	X =  113.445  mm,	Y =   -643.534  mm,	Z =   -257.195  mm,
	W =  90.000 deg,	P =   0.000 deg,	R =   90.000 deg
};
P[2098]{
   GP1:
	UF : 0, UT : 6,		CONFIG : 'N U T, 0, 0, 0',
	X =  119.284  mm,	Y =   -640.249  mm,	Z =   -256.987  mm,
	W =  90.000 deg,	P =   0.000 deg,	R =   90.000 deg
};
P[2099]{
   GP1:
	UF : 0, UT : 6,		CONFIG : 'N U T, 0, 0, 0',
	X =  120.353  mm,	Y =   -639.513  mm,	Z =   -257.274  mm,
	W =  90.000 deg,	P =   0.000 deg,	R =   90.000 deg
};
P[2100]{
   GP1:
	UF : 0, UT : 6,		CONFIG : 'N U T, 0, 0, 0',
	X =  122.366  mm,	Y =   -638.374  mm,	Z =   -257.215  mm,
	W =  90.000 deg,	P =   0.000 deg,	R =   90.000 deg
};
P[2101]{
   GP1:
	UF : 0, UT : 6,		CONFIG : 'N U T, 0, 0, 0',
	X =  125.303  mm,	Y =   -636.720  mm,	Z =   -257.116  mm,
	W =  90.000 deg,	P =   0.000 deg,	R =   90.000 deg
};
P[2102]{
   GP1:
	UF : 0, UT : 6,		CONFIG : 'N U T, 0, 0, 0',
	X =  126.391  mm,	Y =   -636.119  mm,	Z =   -257.049  mm,
	W =  90.000 deg,	P =   0.000 deg,	R =   90.000 deg
};
P[2103]{
   GP1:
	UF : 0, UT : 6,		CONFIG : 'N U T, 0, 0, 0',
	X =  128.149  mm,	Y =   -635.072  mm,	Z =   -257.125  mm,
	W =  90.000 deg,	P =   0.000 deg,	R =   90.000 deg
};
P[2104]{
   GP1:
	UF : 0, UT : 6,		CONFIG : 'N U T, 0, 0, 0',
	X =  129.405  mm,	Y =   -634.261  mm,	Z =   -257.337  mm,
	W =  90.000 deg,	P =   0.000 deg,	R =   90.000 deg
};
P[2105]{
   GP1:
	UF : 0, UT : 6,		CONFIG : 'N U T, 0, 0, 0',
	X =  133.642  mm,	Y =   -631.812  mm,	Z =   -257.340  mm,
	W =  90.000 deg,	P =   0.000 deg,	R =   90.000 deg
};
P[2106]{
   GP1:
	UF : 0, UT : 6,		CONFIG : 'N U T, 0, 0, 0',
	X =  134.817  mm,	Y =   -631.137  mm,	Z =   -257.334  mm,
	W =  90.000 deg,	P =   0.000 deg,	R =   90.000 deg
};
P[2107]{
   GP1:
	UF : 0, UT : 6,		CONFIG : 'N U T, 0, 0, 0',
	X =  135.600  mm,	Y =   -630.719  mm,	Z =   -257.251  mm,
	W =  90.000 deg,	P =   0.000 deg,	R =   90.000 deg
};
P[2108]{
   GP1:
	UF : 0, UT : 6,		CONFIG : 'N U T, 0, 0, 0',
	X =  138.719  mm,	Y =   -628.949  mm,	Z =   -257.176  mm,
	W =  90.000 deg,	P =   0.000 deg,	R =   90.000 deg
};
P[2109]{
   GP1:
	UF : 0, UT : 6,		CONFIG : 'N U T, 0, 0, 0',
	X =  140.494  mm,	Y =   -627.843  mm,	Z =   -257.374  mm,
	W =  90.000 deg,	P =   0.000 deg,	R =   90.000 deg
};
P[2110]{
   GP1:
	UF : 0, UT : 6,		CONFIG : 'N U T, 0, 0, 0',
	X =  144.879  mm,	Y =   -625.464  mm,	Z =   -257.003  mm,
	W =  90.000 deg,	P =   0.000 deg,	R =   90.000 deg
};
P[2111]{
   GP1:
	UF : 0, UT : 6,		CONFIG : 'N U T, 0, 0, 0',
	X =  147.744  mm,	Y =   -623.730  mm,	Z =   -257.195  mm,
	W =  90.000 deg,	P =   0.000 deg,	R =   90.000 deg
};
P[2112]{
   GP1:
	UF : 0, UT : 6,		CONFIG : 'N U T, 0, 0, 0',
	X =  149.698  mm,	Y =   -622.634  mm,	Z =   -257.116  mm,
	W =  90.000 deg,	P =   0.000 deg,	R =   90.000 deg
};
P[2113]{
   GP1:
	UF : 0, UT : 6,		CONFIG : 'N U T, 0, 0, 0',
	X =  150.518  mm,	Y =   -622.121  mm,	Z =   -257.214  mm,
	W =  90.000 deg,	P =   0.000 deg,	R =   90.000 deg
};
P[2114]{
   GP1:
	UF : 0, UT : 6,		CONFIG : 'N U T, 0, 0, 0',
	X =  158.347  mm,	Y =   -617.647  mm,	Z =   -257.099  mm,
	W =  90.000 deg,	P =   0.000 deg,	R =   90.000 deg
};
P[2115]{
   GP1:
	UF : 0, UT : 6,		CONFIG : 'N U T, 0, 0, 0',
	X =  159.078  mm,	Y =   -617.197  mm,	Z =   -257.167  mm,
	W =  90.000 deg,	P =   0.000 deg,	R =   90.000 deg
};
P[2116]{
   GP1:
	UF : 0, UT : 6,		CONFIG : 'N U T, 0, 0, 0',
	X =  160.223  mm,	Y =   -616.456  mm,	Z =   -257.362  mm,
	W =  90.000 deg,	P =   0.000 deg,	R =   90.000 deg
};
P[2117]{
   GP1:
	UF : 0, UT : 6,		CONFIG : 'N U T, 0, 0, 0',
	X =  164.521  mm,	Y =   -614.083  mm,	Z =   -257.100  mm,
	W =  90.000 deg,	P =   0.000 deg,	R =   90.000 deg
};
P[2118]{
   GP1:
	UF : 0, UT : 6,		CONFIG : 'N U T, 0, 0, 0',
	X =  165.339  mm,	Y =   -613.695  mm,	Z =   -256.893  mm,
	W =  90.000 deg,	P =   0.000 deg,	R =   90.000 deg
};
P[2119]{
   GP1:
	UF : 0, UT : 6,		CONFIG : 'N U T, 0, 0, 0',
	X =  166.021  mm,	Y =   -613.178  mm,	Z =   -257.192  mm,
	W =  90.000 deg,	P =   0.000 deg,	R =   90.000 deg
};
P[2120]{
   GP1:
	UF : 0, UT : 6,		CONFIG : 'N U T, 0, 0, 0',
	X =  167.713  mm,	Y =   -612.213  mm,	Z =   -257.164  mm,
	W =  90.000 deg,	P =   0.000 deg,	R =   90.000 deg
};
P[2121]{
   GP1:
	UF : 0, UT : 6,		CONFIG : 'N U T, 0, 0, 0',
	X =  168.696  mm,	Y =   -611.619  mm,	Z =   -257.228  mm,
	W =  90.000 deg,	P =   0.000 deg,	R =   90.000 deg
};
P[2122]{
   GP1:
	UF : 0, UT : 6,		CONFIG : 'N U T, 0, 0, 0',
	X =  169.593  mm,	Y =   -611.059  mm,	Z =   -257.330  mm,
	W =  90.000 deg,	P =   0.000 deg,	R =   90.000 deg
};
P[2123]{
   GP1:
	UF : 0, UT : 6,		CONFIG : 'N U T, 0, 0, 0',
	X =  173.846  mm,	Y =   -608.622  mm,	Z =   -257.287  mm,
	W =  90.000 deg,	P =   0.000 deg,	R =   90.000 deg
};
P[2124]{
   GP1:
	UF : 0, UT : 6,		CONFIG : 'N U T, 0, 0, 0',
	X =  176.233  mm,	Y =   -607.353  mm,	Z =   -257.021  mm,
	W =  90.000 deg,	P =   0.000 deg,	R =   90.000 deg
};
P[2125]{
   GP1:
	UF : 0, UT : 6,		CONFIG : 'N U T, 0, 0, 0',
	X =  179.420  mm,	Y =   -605.394  mm,	Z =   -257.307  mm,
	W =  90.000 deg,	P =   0.000 deg,	R =   90.000 deg
};
P[2126]{
   GP1:
	UF : 0, UT : 6,		CONFIG : 'N U T, 0, 0, 0',
	X =  181.261  mm,	Y =   -604.330  mm,	Z =   -257.311  mm,
	W =  90.000 deg,	P =   0.000 deg,	R =   90.000 deg
};
P[2127]{
   GP1:
	UF : 0, UT : 6,		CONFIG : 'N U T, 0, 0, 0',
	X =  181.963  mm,	Y =   -604.005  mm,	Z =   -257.115  mm,
	W =  90.000 deg,	P =   0.000 deg,	R =   90.000 deg
};
P[2128]{
   GP1:
	UF : 0, UT : 6,		CONFIG : 'N U T, 0, 0, 0',
	X =  184.189  mm,	Y =   -602.626  mm,	Z =   -257.343  mm,
	W =  90.000 deg,	P =   0.000 deg,	R =   90.000 deg
};
P[2129]{
   GP1:
	UF : 0, UT : 6,		CONFIG : 'N U T, 0, 0, 0',
	X =  185.609  mm,	Y =   -601.897  mm,	Z =   -257.124  mm,
	W =  90.000 deg,	P =   0.000 deg,	R =   90.000 deg
};
P[2130]{
   GP1:
	UF : 0, UT : 6,		CONFIG : 'N U T, 0, 0, 0',
	X =  188.140  mm,	Y =   -600.372  mm,	Z =   -257.276  mm,
	W =  90.000 deg,	P =   0.000 deg,	R =   90.000 deg
};
P[2131]{
   GP1:
	UF : 0, UT : 6,		CONFIG : 'N U T, 0, 0, 0',
	X =  191.589  mm,	Y =   -598.356  mm,	Z =   -257.335  mm,
	W =  90.000 deg,	P =   0.000 deg,	R =   90.000 deg
};
P[2132]{
   GP1:
	UF : 0, UT : 6,		CONFIG : 'N U T, 0, 0, 0',
	X =  194.057  mm,	Y =   -596.933  mm,	Z =   -257.332  mm,
	W =  90.000 deg,	P =   0.000 deg,	R =   90.000 deg
};
P[2133]{
   GP1:
	UF : 0, UT : 6,		CONFIG : 'N U T, 0, 0, 0',
	X =  196.582  mm,	Y =   -595.509  mm,	Z =   -257.251  mm,
	W =  90.000 deg,	P =   0.000 deg,	R =   90.000 deg
};
P[2134]{
   GP1:
	UF : 0, UT : 6,		CONFIG : 'N U T, 0, 0, 0',
	X =  198.130  mm,	Y =   -594.683  mm,	Z =   -257.086  mm,
	W =  90.000 deg,	P =   0.000 deg,	R =   90.000 deg
};
P[2135]{
   GP1:
	UF : 0, UT : 6,		CONFIG : 'N U T, 0, 0, 0',
	X =  199.824  mm,	Y =   -593.721  mm,	Z =   -257.048  mm,
	W =  90.000 deg,	P =   0.000 deg,	R =   90.000 deg
};
P[2136]{
   GP1:
	UF : 0, UT : 6,		CONFIG : 'N U T, 0, 0, 0',
	X =  201.772  mm,	Y =   -592.515  mm,	Z =   -257.244  mm,
	W =  90.000 deg,	P =   0.000 deg,	R =   90.000 deg
};
P[2137]{
   GP1:
	UF : 0, UT : 6,		CONFIG : 'N U T, 0, 0, 0',
	X =  203.247  mm,	Y =   -591.664  mm,	Z =   -257.241  mm,
	W =  90.000 deg,	P =   0.000 deg,	R =   90.000 deg
};
P[2138]{
   GP1:
	UF : 0, UT : 6,		CONFIG : 'N U T, 0, 0, 0',
	X =  207.750  mm,	Y =   -589.114  mm,	Z =   -257.121  mm,
	W =  90.000 deg,	P =   0.000 deg,	R =   90.000 deg
};
P[2139]{
   GP1:
	UF : 0, UT : 6,		CONFIG : 'N U T, 0, 0, 0',
	X =  208.446  mm,	Y =   -588.732  mm,	Z =   -257.070  mm,
	W =  90.000 deg,	P =   0.000 deg,	R =   90.000 deg
};
P[2140]{
   GP1:
	UF : 0, UT : 6,		CONFIG : 'N U T, 0, 0, 0',
	X =  210.025  mm,	Y =   -587.832  mm,	Z =   -257.044  mm,
	W =  90.000 deg,	P =   0.000 deg,	R =   90.000 deg
};
P[2141]{
   GP1:
	UF : 0, UT : 6,		CONFIG : 'N U T, 0, 0, 0',
	X =  212.669  mm,	Y =   -586.209  mm,	Z =   -257.278  mm,
	W =  90.000 deg,	P =   0.000 deg,	R =   90.000 deg
};
P[2142]{
   GP1:
	UF : 0, UT : 6,		CONFIG : 'N U T, 0, 0, 0',
	X =  214.485  mm,	Y =   -585.126  mm,	Z =   -257.361  mm,
	W =  90.000 deg,	P =   0.000 deg,	R =   90.000 deg
};
P[2143]{
   GP1:
	UF : 0, UT : 6,		CONFIG : 'N U T, 0, 0, 0',
	X =  215.341  mm,	Y =   -584.730  mm,	Z =   -257.123  mm,
	W =  90.000 deg,	P =   0.000 deg,	R =   90.000 deg
};
P[2144]{
   GP1:
	UF : 0, UT : 6,		CONFIG : 'N U T, 0, 0, 0',
	X =  218.567  mm,	Y =   -582.892  mm,	Z =   -257.063  mm,
	W =  90.000 deg,	P =   0.000 deg,	R =   90.000 deg
};
P[2145]{
   GP1:
	UF : 0, UT : 6,		CONFIG : 'N U T, 0, 0, 0',
	X =  223.016  mm,	Y =   -580.308  mm,	Z =   -257.100  mm,
	W =  90.000 deg,	P =   0.000 deg,	R =   90.000 deg
};
P[2146]{
   GP1:
	UF : 0, UT : 6,		CONFIG : 'N U T, 0, 0, 0',
	X =  223.666  mm,	Y =   -580.001  mm,	Z =   -256.933  mm,
	W =  90.000 deg,	P =   0.000 deg,	R =   90.000 deg
};
P[2147]{
   GP1:
	UF : 0, UT : 6,		CONFIG : 'N U T, 0, 0, 0',
	X =  226.605  mm,	Y =   -578.307  mm,	Z =   -256.925  mm,
	W =  90.000 deg,	P =   0.000 deg,	R =   90.000 deg
};
P[2148]{
   GP1:
	UF : 0, UT : 6,		CONFIG : 'N U T, 0, 0, 0',
	X =  228.043  mm,	Y =   -577.321  mm,	Z =   -257.304  mm,
	W =  90.000 deg,	P =   0.000 deg,	R =   90.000 deg
};
P[2149]{
   GP1:
	UF : 0, UT : 6,		CONFIG : 'N U T, 0, 0, 0',
	X =  228.786  mm,	Y =   -577.012  mm,	Z =   -257.013  mm,
	W =  90.000 deg,	P =   0.000 deg,	R =   90.000 deg
};
P[2150]{
   GP1:
	UF : 0, UT : 6,		CONFIG : 'N U T, 0, 0, 0',
	X =  232.019  mm,	Y =   -575.058  mm,	Z =   -257.225  mm,
	W =  90.000 deg,	P =   0.000 deg,	R =   90.000 deg
};
P[2151]{
   GP1:
	UF : 0, UT : 6,		CONFIG : 'N U T, 0, 0, 0',
	X =  232.928  mm,	Y =   -574.469  mm,	Z =   -257.381  mm,
	W =  90.000 deg,	P =   0.000 deg,	R =   90.000 deg
};
P[2152]{
   GP1:
	UF : 0, UT : 6,		CONFIG : 'N U T, 0, 0, 0',
	X =  235.660  mm,	Y =   -572.931  mm,	Z =   -257.286  mm,
	W =  90.000 deg,	P =   0.000 deg,	R =   90.000 deg
};
P[2153]{
   GP1:
	UF : 0, UT : 6,		CONFIG : 'N U T, 0, 0, 0',
	X =  237.324  mm,	Y =   -572.109  mm,	Z =   -256.947  mm,
	W =  90.000 deg,	P =   0.000 deg,	R =   90.000 deg
};
P[2154]{
   GP1:
	UF : 0, UT : 6,		CONFIG : 'N U T, 0, 0, 0',
	X =  238.722  mm,	Y =   -571.134  mm,	Z =   -257.357  mm,
	W =  90.000 deg,	P =   0.000 deg,	R =   90.000 deg
};
P[2155]{
   GP1:
	UF : 0, UT : 6,		CONFIG : 'N U T, 0, 0, 0',
	X =  242.232  mm,	Y =   -569.250  mm,	Z =   -257.009  mm,
	W =  90.000 deg,	P =   0.000 deg,	R =   90.000 deg
};
P[2156]{
   GP1:
	UF : 0, UT : 6,		CONFIG : 'N U T, 0, 0, 0',
	X =  244.183  mm,	Y =   -567.996  mm,	Z =   -257.322  mm,
	W =  90.000 deg,	P =   0.000 deg,	R =   90.000 deg
};
P[2157]{
   GP1:
	UF : 0, UT : 6,		CONFIG : 'N U T, 0, 0, 0',
	X =  245.455  mm,	Y =   -567.331  mm,	Z =   -257.152  mm,
	W =  90.000 deg,	P =   0.000 deg,	R =   90.000 deg
};
P[2158]{
   GP1:
	UF : 0, UT : 6,		CONFIG : 'N U T, 0, 0, 0',
	X =  246.314  mm,	Y =   -566.740  mm,	Z =   -257.380  mm,
	W =  90.000 deg,	P =   0.000 deg,	R =   90.000 deg
};
P[2159]{
   GP1:
	UF : 0, UT : 6,		CONFIG : 'N U T, 0, 0, 0',
	X =  247.191  mm,	Y =   -566.275  mm,	Z =   -257.279  mm,
	W =  90.000 deg,	P =   0.000 deg,	R =   90.000 deg
};
P[2160]{
   GP1:
	UF : 0, UT : 6,		CONFIG : 'N U T, 0, 0, 0',
	X =  248.158  mm,	Y =   -565.716  mm,	Z =   -257.281  mm,
	W =  90.000 deg,	P =   0.000 deg,	R =   90.000 deg
};
P[2161]{
   GP1:
	UF : 0, UT : 6,		CONFIG : 'N U T, 0, 0, 0',
	X =  250.314  mm,	Y =   -564.475  mm,	Z =   -257.271  mm,
	W =  90.000 deg,	P =   0.000 deg,	R =   90.000 deg
};
P[2162]{
   GP1:
	UF : 0, UT : 6,		CONFIG : 'N U T, 0, 0, 0',
	X =  251.403  mm,	Y =   -563.903  mm,	Z =   -257.135  mm,
	W =  90.000 deg,	P =   0.000 deg,	R =   90.000 deg
};
P[2163]{
   GP1:
	UF : 0, UT : 6,		CONFIG : 'N U T, 0, 0, 0',
	X =  253.414  mm,	Y =   -562.723  mm,	Z =   -257.183  mm,
	W =  90.000 deg,	P =   0.000 deg,	R =   90.000 deg
};
P[2164]{
   GP1:
	UF : 0, UT : 6,		CONFIG : 'N U T, 0, 0, 0',
	X =  259.113  mm,	Y =   -559.505  mm,	Z =   -257.004  mm,
	W =  90.000 deg,	P =   0.000 deg,	R =   90.000 deg
};
P[2165]{
   GP1:
	UF : 0, UT : 6,		CONFIG : 'N U T, 0, 0, 0',
	X =  261.683  mm,	Y =   -557.964  mm,	Z =   -257.143  mm,
	W =  90.000 deg,	P =   0.000 deg,	R =   90.000 deg
};
P[2166]{
   GP1:
	UF : 0, UT : 6,		CONFIG : 'N U T, 0, 0, 0',
	X =  262.661  mm,	Y =   -557.339  mm,	Z =   -257.291  mm,
	W =  90.000 deg,	P =   0.000 deg,	R =   90.000 deg
};
P[2167]{
   GP1:
	UF : 0, UT : 6,		CONFIG : 'N U T, 0, 0, 0',
	X =  263.771  mm,	Y =   -556.827  mm,	Z =   -256.978  mm,
	W =  90.000 deg,	P =   0.000 deg,	R =   90.000 deg
};
P[2168]{
   GP1:
	UF : 0, UT : 6,		CONFIG : 'N U T, 0, 0, 0',
	X =  266.090  mm,	Y =   -555.345  mm,	Z =   -257.325  mm,
	W =  90.000 deg,	P =   0.000 deg,	R =   90.000 deg
};
P[2169]{
   GP1:
	UF : 0, UT : 6,		CONFIG : 'N U T, 0, 0, 0',
	X =  266.938  mm,	Y =   -555.016  mm,	Z =   -256.934  mm,
	W =  90.000 deg,	P =   0.000 deg,	R =   90.000 deg
};
P[2170]{
   GP1:
	UF : 0, UT : 6,		CONFIG : 'N U T, 0, 0, 0',
	X =  270.560  mm,	Y =   -552.768  mm,	Z =   -257.316  mm,
	W =  90.000 deg,	P =   0.000 deg,	R =   90.000 deg
};
P[2171]{
   GP1:
	UF : 0, UT : 6,		CONFIG : 'N U T, 0, 0, 0',
	X =  272.010  mm,	Y =   -551.959  mm,	Z =   -257.248  mm,
	W =  90.000 deg,	P =   0.000 deg,	R =   90.000 deg
};
P[2172]{
   GP1:
	UF : 0, UT : 6,		CONFIG : 'N U T, 0, 0, 0',
	X =  273.469  mm,	Y =   -551.079  mm,	Z =   -257.337  mm,
	W =  90.000 deg,	P =   0.000 deg,	R =   90.000 deg
};
P[2173]{
   GP1:
	UF : 0, UT : 6,		CONFIG : 'N U T, 0, 0, 0',
	X =  277.285  mm,	Y =   -548.933  mm,	Z =   -257.198  mm,
	W =  90.000 deg,	P =   0.000 deg,	R =   90.000 deg
};
P[2174]{
   GP1:
	UF : 0, UT : 6,		CONFIG : 'N U T, 0, 0, 0',
	X =  280.570  mm,	Y =   -546.991  mm,	Z =   -257.309  mm,
	W =  90.000 deg,	P =   0.000 deg,	R =   90.000 deg
};
P[2175]{
   GP1:
	UF : 0, UT : 6,		CONFIG : 'N U T, 0, 0, 0',
	X =  282.214  mm,	Y =   -546.154  mm,	Z =   -257.036  mm,
	W =  90.000 deg,	P =   0.000 deg,	R =   90.000 deg
};
P[2176]{
   GP1:
	UF : 0, UT : 6,		CONFIG : 'N U T, 0, 0, 0',
	X =  284.085  mm,	Y =   -544.962  mm,	Z =   -257.306  mm,
	W =  90.000 deg,	P =   0.000 deg,	R =   90.000 deg
};
P[2177]{
   GP1:
	UF : 0, UT : 6,		CONFIG : 'N U T, 0, 0, 0',
	X =  286.474  mm,	Y =   -543.555  mm,	Z =   -257.373  mm,
	W =  90.000 deg,	P =   0.000 deg,	R =   90.000 deg
};
P[2178]{
   GP1:
	UF : 0, UT : 6,		CONFIG : 'N U T, 0, 0, 0',
	X =  288.966  mm,	Y =   -542.236  mm,	Z =   -257.081  mm,
	W =  90.000 deg,	P =   0.000 deg,	R =   90.000 deg
};
P[2179]{
   GP1:
	UF : 0, UT : 6,		CONFIG : 'N U T, 0, 0, 0',
	X =  292.153  mm,	Y =   -540.456  mm,	Z =   -256.936  mm,
	W =  90.000 deg,	P =   0.000 deg,	R =   90.000 deg
};
P[2180]{
   GP1:
	UF : 0, UT : 6,		CONFIG : 'N U T, 0, 0, 0',
	X =  299.062  mm,	Y =   -536.298  mm,	Z =   -257.346  mm,
	W =  90.000 deg,	P =   0.000 deg,	R =   90.000 deg
};
P[2181]{
   GP1:
	UF : 0, UT : 6,		CONFIG : 'N U T, 0, 0, 0',
	X =  299.968  mm,	Y =   -535.760  mm,	Z =   -257.381  mm,
	W =  90.000 deg,	P =   0.000 deg,	R =   90.000 deg
};
P[2182]{
   GP1:
	UF : 0, UT : 6,		CONFIG : 'N U T, 0, 0, 0',
	X =  300.824  mm,	Y =   -535.320  mm,	Z =   -257.251  mm,
	W =  90.000 deg,	P =   0.000 deg,	R =   90.000 deg
};
P[2183]{
   GP1:
	UF : 0, UT : 6,		CONFIG : 'N U T, 0, 0, 0',
	X =  301.911  mm,	Y =   -534.684  mm,	Z =   -257.272  mm,
	W =  90.000 deg,	P =   0.000 deg,	R =   90.000 deg
};
P[2184]{
   GP1:
	UF : 0, UT : 6,		CONFIG : 'N U T, 0, 0, 0',
	X =  305.019  mm,	Y =   -532.905  mm,	Z =   -257.233  mm,
	W =  90.000 deg,	P =   0.000 deg,	R =   90.000 deg
};
P[2185]{
   GP1:
	UF : 0, UT : 6,		CONFIG : 'N U T, 0, 0, 0',
	X =  307.325  mm,	Y =   -531.551  mm,	Z =   -257.287  mm,
	W =  90.000 deg,	P =   0.000 deg,	R =   90.000 deg
};
P[2186]{
   GP1:
	UF : 0, UT : 6,		CONFIG : 'N U T, 0, 0, 0',
	X =  309.546  mm,	Y =   -530.345  mm,	Z =   -257.103  mm,
	W =  90.000 deg,	P =   0.000 deg,	R =   90.000 deg
};
P[2187]{
   GP1:
	UF : 0, UT : 6,		CONFIG : 'N U T, 0, 0, 0',
	X =  311.447  mm,	Y =   -529.152  mm,	Z =   -257.334  mm,
	W =  90.000 deg,	P =   0.000 deg,	R =   90.000 deg
};
P[2188]{
   GP1:
	UF : 0, UT : 6,		CONFIG : 'N U T, 0, 0, 0',
	X =  314.729  mm,	Y =   -527.268  mm,	Z =   -257.306  mm,
	W =  90.000 deg,	P =   0.000 deg,	R =   90.000 deg
};
P[2189]{
   GP1:
	UF : 0, UT : 6,		CONFIG : 'N U T, 0, 0, 0',
	X =  316.875  mm,	Y =   -526.069  mm,	Z =   -257.211  mm,
	W =  90.000 deg,	P =   0.000 deg,	R =   90.000 deg
};
P[2190]{
   GP1:
	UF : 0, UT : 6,		CONFIG : 'N U T, 0, 0, 0',
	X =  318.015  mm,	Y =   -525.355  mm,	Z =   -257.345  mm,
	W =  90.000 deg,	P =   0.000 deg,	R =   90.000 deg
};
P[2191]{
   GP1:
	UF : 0, UT : 6,		CONFIG : 'N U T, 0, 0, 0',
	X =  318.649  mm,	Y =   -525.057  mm,	Z =   -257.180  mm,
	W =  90.000 deg,	P =   0.000 deg,	R =   90.000 deg
};
P[2192]{
   GP1:
	UF : 0, UT : 6,		CONFIG : 'N U T, 0, 0, 0',
	X =  322.343  mm,	Y =   -522.958  mm,	Z =   -257.099  mm,
	W =  90.000 deg,	P =   0.000 deg,	R =   90.000 deg
};
P[2193]{
   GP1:
	UF : 0, UT : 6,		CONFIG : 'N U T, 0, 0, 0',
	X =  322.941  mm,	Y =   -522.528  mm,	Z =   -257.305  mm,
	W =  90.000 deg,	P =   0.000 deg,	R =   90.000 deg
};
P[2194]{
   GP1:
	UF : 0, UT : 6,		CONFIG : 'N U T, 0, 0, 0',
	X =  324.717  mm,	Y =   -521.576  mm,	Z =   -257.127  mm,
	W =  90.000 deg,	P =   0.000 deg,	R =   90.000 deg
};
P[2195]{
   GP1:
	UF : 0, UT : 6,		CONFIG : 'N U T, 0, 0, 0',
	X =  327.318  mm,	Y =   -520.012  mm,	Z =   -257.277  mm,
	W =  90.000 deg,	P =   0.000 deg,	R =   90.000 deg
};
P[2196]{
   GP1:
	UF : 0, UT : 6,		CONFIG : 'N U T, 0, 0, 0',
	X =  329.668  mm,	Y =   -518.723  mm,	Z =   -257.112  mm,
	W =  90.000 deg,	P =   0.000 deg,	R =   90.000 deg
};
P[2197]{
   GP1:
	UF : 0, UT : 6,		CONFIG : 'N U T, 0, 0, 0',
	X =  331.747  mm,	Y =   -517.451  mm,	Z =   -257.286  mm,
	W =  90.000 deg,	P =   0.000 deg,	R =   90.000 deg
};
P[2198]{
   GP1:
	UF : 0, UT : 6,		CONFIG : 'N U T, 0, 0, 0',
	X =  335.566  mm,	Y =   -515.313  mm,	Z =   -257.124  mm,
	W =  90.000 deg,	P =   0.000 deg,	R =   90.000 deg
};
P[2199]{
   GP1:
	UF : 0, UT : 6,		CONFIG : 'N U T, 0, 0, 0',
	X =  337.324  mm,	Y =   -514.263  mm,	Z =   -257.209  mm,
	W =  90.000 deg,	P =   0.000 deg,	R =   90.000 deg
};
P[2200]{
   GP1:
	UF : 0, UT : 6,		CONFIG : 'N U T, 0, 0, 0',
	X =  338.434  mm,	Y =   -513.597  mm,	Z =   -257.269  mm,
	W =  90.000 deg,	P =   0.000 deg,	R =   90.000 deg
};
P[2201]{
   GP1:
	UF : 0, UT : 6,		CONFIG : 'N U T, 0, 0, 0',
	X =  340.084  mm,	Y =   -512.599  mm,	Z =   -257.377  mm,
	W =  90.000 deg,	P =   0.000 deg,	R =   90.000 deg
};
P[2202]{
   GP1:
	UF : 0, UT : 6,		CONFIG : 'N U T, 0, 0, 0',
	X =  342.231  mm,	Y =   -511.494  mm,	Z =   -257.053  mm,
	W =  90.000 deg,	P =   0.000 deg,	R =   90.000 deg
};
P[2203]{
   GP1:
	UF : 0, UT : 6,		CONFIG : 'N U T, 0, 0, 0',
	X =  344.018  mm,	Y =   -510.380  mm,	Z =   -257.251  mm,
	W =  90.000 deg,	P =   0.000 deg,	R =   90.000 deg
};
P[2204]{
   GP1:
	UF : 0, UT : 6,		CONFIG : 'N U T, 0, 0, 0',
	X =  346.852  mm,	Y =   -508.709  mm,	Z =   -257.335  mm,
	W =  90.000 deg,	P =   0.000 deg,	R =   90.000 deg
};
P[2205]{
   GP1:
	UF : 0, UT : 6,		CONFIG : 'N U T, 0, 0, 0',
	X =  348.451  mm,	Y =   -507.914  mm,	Z =   -257.024  mm,
	W =  90.000 deg,	P =   0.000 deg,	R =   90.000 deg
};
P[2206]{
   GP1:
	UF : 0, UT : 6,		CONFIG : 'N U T, 0, 0, 0',
	X =  354.237  mm,	Y =   -504.581  mm,	Z =   -257.005  mm,
	W =  90.000 deg,	P =   0.000 deg,	R =   90.000 deg
};
P[2207]{
   GP1:
	UF : 0, UT : 6,		CONFIG : 'N U T, 0, 0, 0',
	X =  356.023  mm,	Y =   -503.535  mm,	Z =   -257.042  mm,
	W =  90.000 deg,	P =   0.000 deg,	R =   90.000 deg
};
P[2208]{
   GP1:
	UF : 0, UT : 6,		CONFIG : 'N U T, 0, 0, 0',
	X =  357.474  mm,	Y =   -502.737  mm,	Z =   -256.944  mm,
	W =  90.000 deg,	P =   0.000 deg,	R =   90.000 deg
};
P[2209]{
   GP1:
	UF : 0, UT : 6,		CONFIG : 'N U T, 0, 0, 0',
	X =  358.347  mm,	Y =   -502.088  mm,	Z =   -257.296  mm,
	W =  90.000 deg,	P =   0.000 deg,	R =   90.000 deg
};
P[2210]{
   GP1:
	UF : 0, UT : 6,		CONFIG : 'N U T, 0, 0, 0',
	X =  361.299  mm,	Y =   -500.366  mm,	Z =   -257.340  mm,
	W =  90.000 deg,	P =   0.000 deg,	R =   90.000 deg
};
P[2211]{
   GP1:
	UF : 0, UT : 6,		CONFIG : 'N U T, 0, 0, 0',
	X =  365.272  mm,	Y =   -498.145  mm,	Z =   -257.163  mm,
	W =  90.000 deg,	P =   0.000 deg,	R =   90.000 deg
};
P[2212]{
   GP1:
	UF : 0, UT : 6,		CONFIG : 'N U T, 0, 0, 0',
	X =  367.462  mm,	Y =   -496.906  mm,	Z =   -257.102  mm,
	W =  90.000 deg,	P =   0.000 deg,	R =   90.000 deg
};
P[2213]{
   GP1:
	UF : 0, UT : 6,		CONFIG : 'N U T, 0, 0, 0',
	X =  369.304  mm,	Y =   -495.901  mm,	Z =   -256.958  mm,
	W =  90.000 deg,	P =   0.000 deg,	R =   90.000 deg
};
P[2214]{
   GP1:
	UF : 0, UT : 6,		CONFIG : 'N U T, 0, 0, 0',
	X =  372.314  mm,	Y =   -494.181  mm,	Z =   -256.916  mm,
	W =  90.000 deg,	P =   0.000 deg,	R =   90.000 deg
};
P[2215]{
   GP1:
	UF : 0, UT : 6,		CONFIG : 'N U T, 0, 0, 0',
	X =  374.415  mm,	Y =   -492.809  mm,	Z =   -257.300  mm,
	W =  90.000 deg,	P =   0.000 deg,	R =   90.000 deg
};
P[2216]{
   GP1:
	UF : 0, UT : 6,		CONFIG : 'N U T, 0, 0, 0',
	X =  376.903  mm,	Y =   -491.366  mm,	Z =   -257.314  mm,
	W =  90.000 deg,	P =   0.000 deg,	R =   90.000 deg
};
P[2217]{
   GP1:
	UF : 0, UT : 6,		CONFIG : 'N U T, 0, 0, 0',
	X =  378.917  mm,	Y =   -490.208  mm,	Z =   -257.302  mm,
	W =  90.000 deg,	P =   0.000 deg,	R =   90.000 deg
};
P[2218]{
   GP1:
	UF : 0, UT : 6,		CONFIG : 'N U T, 0, 0, 0',
	X =  382.035  mm,	Y =   -488.470  mm,	Z =   -257.155  mm,
	W =  90.000 deg,	P =   0.000 deg,	R =   90.000 deg
};
P[2219]{
   GP1:
	UF : 0, UT : 6,		CONFIG : 'N U T, 0, 0, 0',
	X =  385.243  mm,	Y =   -486.688  mm,	Z =   -256.981  mm,
	W =  90.000 deg,	P =   0.000 deg,	R =   90.000 deg
};
P[2220]{
   GP1:
	UF : 0, UT : 6,		CONFIG : 'N U T, 0, 0, 0',
	X =  387.116  mm,	Y =   -485.459  mm,	Z =   -257.340  mm,
	W =  90.000 deg,	P =   0.000 deg,	R =   90.000 deg
};
P[2221]{
   GP1:
	UF : 0, UT : 6,		CONFIG : 'N U T, 0, 0, 0',
	X =  389.384  mm,	Y =   -484.194  mm,	Z =   -257.233  mm,
	W =  90.000 deg,	P =   0.000 deg,	R =   90.000 deg
};
P[2222]{
   GP1:
	UF : 0, UT : 6,		CONFIG : 'N U T, 0, 0, 0',
	X =  392.428  mm,	Y =   -482.573  mm,	Z =   -256.902  mm,
	W =  90.000 deg,	P =   0.000 deg,	R =   90.000 deg
};
P[2223]{
   GP1:
	UF : 0, UT : 6,		CONFIG : 'N U T, 0, 0, 0',
	X =  394.034  mm,	Y =   -481.475  mm,	Z =   -257.315  mm,
	W =  90.000 deg,	P =   0.000 deg,	R =   90.000 deg
};
P[2224]{
   GP1:
	UF : 0, UT : 6,		CONFIG : 'N U T, 0, 0, 0',
	X =  398.186  mm,	Y =   -479.056  mm,	Z =   -257.368  mm,
	W =  90.000 deg,	P =   0.000 deg,	R =   90.000 deg
};
P[2225]{
   GP1:
	UF : 0, UT : 6,		CONFIG : 'N U T, 0, 0, 0',
	X =  399.076  mm,	Y =   -478.680  mm,	Z =   -257.032  mm,
	W =  90.000 deg,	P =   0.000 deg,	R =   90.000 deg
};
P[2226]{
   GP1:
	UF : 0, UT : 6,		CONFIG : 'N U T, 0, 0, 0',
	X =  403.801  mm,	Y =   -475.854  mm,	Z =   -257.268  mm,
	W =  90.000 deg,	P =   0.000 deg,	R =   90.000 deg
};
P[2227]{
   GP1:
	UF : 0, UT : 6,		CONFIG : 'N U T, 0, 0, 0',
	X =  404.435  mm,	Y =   -475.476  mm,	Z =   -257.300  mm,
	W =  90.000 deg,	P =   0.000 deg,	R =   90.000 deg
};
P[2228]{
   GP1:
	UF : 0, UT : 6,		CONFIG : 'N U T, 0, 0, 0',
	X =  405.253  mm,	Y =   -475.133  mm,	Z =   -256.986  mm,
	W =  90.000 deg,	P =   0.000 deg,	R =   90.000 deg
};
P[2229]{
   GP1:
	UF : 0, UT : 6,		CONFIG : 'N U T, 0, 0, 0',
	X =  407.120  mm,	Y =   -474.036  mm,	Z =   -257.034  mm,
	W =  90.000 deg,	P =   0.000 deg,	R =   90.000 deg
};
P[2230]{
   GP1:
	UF : 0, UT : 6,		CONFIG : 'N U T, 0, 0, 0',
	X =  408.408  mm,	Y =   -473.148  mm,	Z =   -257.382  mm,
	W =  90.000 deg,	P =   0.000 deg,	R =   90.000 deg
};
P[2231]{
   GP1:
	UF : 0, UT : 6,		CONFIG : 'N U T, 0, 0, 0',
	X =  411.863  mm,	Y =   -471.269  mm,	Z =   -257.101  mm,
	W =  90.000 deg,	P =   0.000 deg,	R =   90.000 deg
};
P[2232]{
   GP1:
	UF : 0, UT : 6,		CONFIG : 'N U T, 0, 0, 0',
	X =  414.660  mm,	Y =   -469.730  mm,	Z =   -256.918  mm,
	W =  90.000 deg,	P =   0.000 deg,	R =   90.000 deg
};
P[2233]{
   GP1:
	UF : 0, UT : 6,		CONFIG : 'N U T, 0, 0, 0',
	X =  415.293  mm,	Y =   -469.272  mm,	Z =   -257.139  mm,
	W =  90.000 deg,	P =   0.000 deg,	R =   90.000 deg
};
P[2234]{
   GP1:
	UF : 0, UT : 6,		CONFIG : 'N U T, 0, 0, 0',
	X =  416.370  mm,	Y =   -468.613  mm,	Z =   -257.231  mm,
	W =  90.000 deg,	P =   0.000 deg,	R =   90.000 deg
};
P[2235]{
   GP1:
	UF : 0, UT : 6,		CONFIG : 'N U T, 0, 0, 0',
	X =  422.087  mm,	Y =   -465.404  mm,	Z =   -257.007  mm,
	W =  90.000 deg,	P =   0.000 deg,	R =   90.000 deg
};
P[2236]{
   GP1:
	UF : 0, UT : 6,		CONFIG : 'N U T, 0, 0, 0',
	X =  423.943  mm,	Y =   -464.184  mm,	Z =   -257.367  mm,
	W =  90.000 deg,	P =   0.000 deg,	R =   90.000 deg
};
P[2237]{
   GP1:
	UF : 0, UT : 6,		CONFIG : 'N U T, 0, 0, 0',
	X =  424.656  mm,	Y =   -463.783  mm,	Z =   -257.344  mm,
	W =  90.000 deg,	P =   0.000 deg,	R =   90.000 deg
};
P[2238]{
   GP1:
	UF : 0, UT : 6,		CONFIG : 'N U T, 0, 0, 0',
	X =  426.200  mm,	Y =   -462.965  mm,	Z =   -257.164  mm,
	W =  90.000 deg,	P =   0.000 deg,	R =   90.000 deg
};
P[2239]{
   GP1:
	UF : 0, UT : 6,		CONFIG : 'N U T, 0, 0, 0',
	X =  429.821  mm,	Y =   -460.976  mm,	Z =   -256.919  mm,
	W =  90.000 deg,	P =   0.000 deg,	R =   90.000 deg
};
P[2240]{
   GP1:
	UF : 0, UT : 6,		CONFIG : 'N U T, 0, 0, 0',
	X =  430.662  mm,	Y =   -460.337  mm,	Z =   -257.288  mm,
	W =  90.000 deg,	P =   0.000 deg,	R =   90.000 deg
};
P[2241]{
   GP1:
	UF : 0, UT : 6,		CONFIG : 'N U T, 0, 0, 0',
	X =  431.850  mm,	Y =   -459.710  mm,	Z =   -257.147  mm,
	W =  90.000 deg,	P =   0.000 deg,	R =   90.000 deg
};
P[2242]{
   GP1:
	UF : 0, UT : 6,		CONFIG : 'N U T, 0, 0, 0',
	X =  435.083  mm,	Y =   -457.856  mm,	Z =   -257.115  mm,
	W =  90.000 deg,	P =   0.000 deg,	R =   90.000 deg
};
P[2243]{
   GP1:
	UF : 0, UT : 6,		CONFIG : 'N U T, 0, 0, 0',
	X =  435.759  mm,	Y =   -457.389  mm,	Z =   -257.302  mm,
	W =  90.000 deg,	P =   0.000 deg,	R =   90.000 deg
};
P[2244]{
   GP1:
	UF : 0, UT : 6,		CONFIG : 'N U T, 0, 0, 0',
	X =  437.736  mm,	Y =   -456.303  mm,	Z =   -257.166  mm,
	W =  90.000 deg,	P =   0.000 deg,	R =   90.000 deg
};
P[2245]{
   GP1:
	UF : 0, UT : 6,		CONFIG : 'N U T, 0, 0, 0',
	X =  438.883  mm,	Y =   -455.551  mm,	Z =   -257.385  mm,
	W =  90.000 deg,	P =   0.000 deg,	R =   90.000 deg
};
P[2246]{
   GP1:
	UF : 0, UT : 6,		CONFIG : 'N U T, 0, 0, 0',
	X =  440.632  mm,	Y =   -454.645  mm,	Z =   -257.131  mm,
	W =  90.000 deg,	P =   0.000 deg,	R =   90.000 deg
};
P[2247]{
   GP1:
	UF : 0, UT : 6,		CONFIG : 'N U T, 0, 0, 0',
	X =  445.039  mm,	Y =   -452.131  mm,	Z =   -257.059  mm,
	W =  90.000 deg,	P =   0.000 deg,	R =   90.000 deg
};
P[2248]{
   GP1:
	UF : 0, UT : 6,		CONFIG : 'N U T, 0, 0, 0',
	X =  445.777  mm,	Y =   -451.600  mm,	Z =   -257.313  mm,
	W =  90.000 deg,	P =   0.000 deg,	R =   90.000 deg
};
P[2249]{
   GP1:
	UF : 0, UT : 6,		CONFIG : 'N U T, 0, 0, 0',
	X =  449.490  mm,	Y =   -449.518  mm,	Z =   -257.161  mm,
	W =  90.000 deg,	P =   0.000 deg,	R =   90.000 deg
};
P[2250]{
   GP1:
	UF : 0, UT : 6,		CONFIG : 'N U T, 0, 0, 0',
	X =  450.101  mm,	Y =   -449.138  mm,	Z =   -257.227  mm,
	W =  90.000 deg,	P =   0.000 deg,	R =   90.000 deg
};
P[2251]{
   GP1:
	UF : 0, UT : 6,		CONFIG : 'N U T, 0, 0, 0',
	X =  454.075  mm,	Y =   -446.925  mm,	Z =   -257.029  mm,
	W =  90.000 deg,	P =   0.000 deg,	R =   90.000 deg
};
P[2252]{
   GP1:
	UF : 0, UT : 6,		CONFIG : 'N U T, 0, 0, 0',
	X =  455.112  mm,	Y =   -446.282  mm,	Z =   -257.137  mm,
	W =  90.000 deg,	P =   0.000 deg,	R =   90.000 deg
};
P[2253]{
   GP1:
	UF : 0, UT : 6,		CONFIG : 'N U T, 0, 0, 0',
	X =  459.811  mm,	Y =   -443.526  mm,	Z =   -257.243  mm,
	W =  90.000 deg,	P =   0.000 deg,	R =   90.000 deg
};
P[2254]{
   GP1:
	UF : 0, UT : 6,		CONFIG : 'N U T, 0, 0, 0',
	X =  460.758  mm,	Y =   -443.019  mm,	Z =   -257.146  mm,
	W =  90.000 deg,	P =   0.000 deg,	R =   90.000 deg
};
P[2255]{
   GP1:
	UF : 0, UT : 6,		CONFIG : 'N U T, 0, 0, 0',
	X =  462.036  mm,	Y =   -442.186  mm,	Z =   -257.377  mm,
	W =  90.000 deg,	P =   0.000 deg,	R =   90.000 deg
};
P[2256]{
   GP1:
	UF : 0, UT : 6,		CONFIG : 'N U T, 0, 0, 0',
	X =  465.885  mm,	Y =   -439.972  mm,	Z =   -257.357  mm,
	W =  90.000 deg,	P =   0.000 deg,	R =   90.000 deg
};
P[2257]{
   GP1:
	UF : 0, UT : 6,		CONFIG : 'N U T, 0, 0, 0',
	X =  468.570  mm,	Y =   -438.410  mm,	Z =   -257.385  mm,
	W =  90.000 deg,	P =   0.000 deg,	R =   90.000 deg
};
P[2258]{
   GP1:
	UF : 0, UT : 6,		CONFIG : 'N U T, 0, 0, 0',
	X =  469.575  mm,	Y =   -437.990  mm,	Z =   -256.995  mm,
	W =  90.000 deg,	P =   0.000 deg,	R =   90.000 deg
};
P[2259]{
   GP1:
	UF : 0, UT : 6,		CONFIG : 'N U T, 0, 0, 0',
	X =  470.439  mm,	Y =   -437.428  mm,	Z =   -257.148  mm,
	W =  90.000 deg,	P =   0.000 deg,	R =   90.000 deg
};
P[2260]{
   GP1:
	UF : 0, UT : 6,		CONFIG : 'N U T, 0, 0, 0',
	X =  475.724  mm,	Y =   -434.380  mm,	Z =   -257.141  mm,
	W =  90.000 deg,	P =   0.000 deg,	R =   90.000 deg
};
P[2261]{
   GP1:
	UF : 0, UT : 6,		CONFIG : 'N U T, 0, 0, 0',
	X =  476.291  mm,	Y =   -433.962  mm,	Z =   -257.360  mm,
	W =  90.000 deg,	P =   0.000 deg,	R =   90.000 deg
};
P[2262]{
   GP1:
	UF : 0, UT : 6,		CONFIG : 'N U T, 0, 0, 0',
	X =  478.577  mm,	Y =   -432.802  mm,	Z =   -256.973  mm,
	W =  90.000 deg,	P =   0.000 deg,	R =   90.000 deg
};
P[2263]{
   GP1:
	UF : 0, UT : 6,		CONFIG : 'N U T, 0, 0, 0',
	X =  479.292  mm,	Y =   -432.293  mm,	Z =   -257.206  mm,
	W =  90.000 deg,	P =   0.000 deg,	R =   90.000 deg
};
P[2264]{
   GP1:
	UF : 0, UT : 6,		CONFIG : 'N U T, 0, 0, 0',
	X =  483.302  mm,	Y =   -429.916  mm,	Z =   -257.353  mm,
	W =  90.000 deg,	P =   0.000 deg,	R =   90.000 deg
};
P[2265]{
   GP1:
	UF : 0, UT : 6,		CONFIG : 'N U T, 0, 0, 0',
	X =  484.058  mm,	Y =   -429.649  mm,	Z =   -256.943  mm,
	W =  90.000 deg,	P =   0.000 deg,	R =   90.000 deg
};
P[2266]{
   GP1:
	UF : 0, UT : 6,		CONFIG : 'N U T, 0, 0, 0',
	X =  487.753  mm,	Y =   -427.407  mm,	Z =   -257.205  mm,
	W =  90.000 deg,	P =   0.000 deg,	R =   90.000 deg
};
P[2267]{
   GP1:
	UF : 0, UT : 6,		CONFIG : 'N U T, 0, 0, 0',
	X =  488.970  mm,	Y =   -426.742  mm,	Z =   -257.115  mm,
	W =  90.000 deg,	P =   0.000 deg,	R =   90.000 deg
};
P[2268]{
   GP1:
	UF : 0, UT : 6,		CONFIG : 'N U T, 0, 0, 0',
	X =  491.365  mm,	Y =   -425.353  mm,	Z =   -257.129  mm,
	W =  90.000 deg,	P =   0.000 deg,	R =   90.000 deg
};
P[2269]{
   GP1:
	UF : 0, UT : 6,		CONFIG : 'N U T, 0, 0, 0',
	X =  493.299  mm,	Y =   -424.291  mm,	Z =   -257.000  mm,
	W =  90.000 deg,	P =   0.000 deg,	R =   90.000 deg
};
P[2270]{
   GP1:
	UF : 0, UT : 6,		CONFIG : 'N U T, 0, 0, 0',
	X =  494.109  mm,	Y =   -423.674  mm,	Z =   -257.361  mm,
	W =  90.000 deg,	P =   0.000 deg,	R =   90.000 deg
};
P[2271]{
   GP1:
	UF : 0, UT : 6,		CONFIG : 'N U T, 0, 0, 0',
	X =  499.841  mm,	Y =   -420.463  mm,	Z =   -257.121  mm,
	W =  90.000 deg,	P =   0.000 deg,	R =   90.000 deg
};
P[2272]{
   GP1:
	UF : 0, UT : 6,		CONFIG : 'N U T, 0, 0, 0',
	X =  501.890  mm,	Y =   -419.186  mm,	Z =   -257.349  mm,
	W =  90.000 deg,	P =   0.000 deg,	R =   90.000 deg
};
P[2273]{
   GP1:
	UF : 0, UT : 6,		CONFIG : 'N U T, 0, 0, 0',
	X =  507.068  mm,	Y =   -416.277  mm,	Z =   -257.153  mm,
	W =  90.000 deg,	P =   0.000 deg,	R =   90.000 deg
};
P[2274]{
   GP1:
	UF : 0, UT : 6,		CONFIG : 'N U T, 0, 0, 0',
	X =  507.694  mm,	Y =   -415.876  mm,	Z =   -257.250  mm,
	W =  90.000 deg,	P =   0.000 deg,	R =   90.000 deg
};
P[2275]{
   GP1:
	UF : 0, UT : 6,		CONFIG : 'N U T, 0, 0, 0',
	X =  510.587  mm,	Y =   -414.332  mm,	Z =   -256.942  mm,
	W =  90.000 deg,	P =   0.000 deg,	R =   90.000 deg
};
P[2276]{
   GP1:
	UF : 0, UT : 6,		CONFIG : 'N U T, 0, 0, 0',
	X =  511.136  mm,	Y =   -413.834  mm,	Z =   -257.381  mm,
	W =  90.000 deg,	P =   0.000 deg,	R =   90.000 deg
};
P[2277]{
   GP1:
	UF : 0, UT : 6,		CONFIG : 'N U T, 0, 0, 0',
	X =  512.108  mm,	Y =   -413.415  mm,	Z =   -257.034  mm,
	W =  90.000 deg,	P =   0.000 deg,	R =   90.000 deg
};
P[2278]{
   GP1:
	UF : 0, UT : 6,		CONFIG : 'N U T, 0, 0, 0',
	X =  513.207  mm,	Y =   -412.674  mm,	Z =   -257.294  mm,
	W =  90.000 deg,	P =   0.000 deg,	R =   90.000 deg
};
P[2279]{
   GP1:
	UF : 0, UT : 6,		CONFIG : 'N U T, 0, 0, 0',
	X =  515.155  mm,	Y =   -411.642  mm,	Z =   -257.070  mm,
	W =  90.000 deg,	P =   0.000 deg,	R =   90.000 deg
};
P[2280]{
   GP1:
	UF : 0, UT : 6,		CONFIG : 'N U T, 0, 0, 0',
	X =  516.066  mm,	Y =   -411.050  mm,	Z =   -257.229  mm,
	W =  90.000 deg,	P =   0.000 deg,	R =   90.000 deg
};
P[2281]{
   GP1:
	UF : 0, UT : 6,		CONFIG : 'N U T, 0, 0, 0',
	X =  517.720  mm,	Y =   -410.073  mm,	Z =   -257.283  mm,
	W =  90.000 deg,	P =   0.000 deg,	R =   90.000 deg
};
P[2282]{
   GP1:
	UF : 0, UT : 6,		CONFIG : 'N U T, 0, 0, 0',
	X =  521.089  mm,	Y =   -408.242  mm,	Z =   -257.005  mm,
	W =  90.000 deg,	P =   0.000 deg,	R =   90.000 deg
};
P[2283]{
   GP1:
	UF : 0, UT : 6,		CONFIG : 'N U T, 0, 0, 0',
	X =  521.760  mm,	Y =   -407.711  mm,	Z =   -257.354  mm,
	W =  90.000 deg,	P =   0.000 deg,	R =   90.000 deg
};
P[2284]{
   GP1:
	UF : 0, UT : 6,		CONFIG : 'N U T, 0, 0, 0',
	X =  523.006  mm,	Y =   -407.132  mm,	Z =   -257.015  mm,
	W =  90.000 deg,	P =   0.000 deg,	R =   90.000 deg
};
P[2285]{
   GP1:
	UF : 0, UT : 6,		CONFIG : 'N U T, 0, 0, 0',
	X =  523.908  mm,	Y =   -406.503  mm,	Z =   -257.277  mm,
	W =  90.000 deg,	P =   0.000 deg,	R =   90.000 deg
};
P[2286]{
   GP1:
	UF : 0, UT : 6,		CONFIG : 'N U T, 0, 0, 0',
	X =  526.832  mm,	Y =   -404.832  mm,	Z =   -257.234  mm,
	W =  90.000 deg,	P =   0.000 deg,	R =   90.000 deg
};
P[2287]{
   GP1:
	UF : 0, UT : 6,		CONFIG : 'N U T, 0, 0, 0',
	X =  527.918  mm,	Y =   -404.221  mm,	Z =   -257.194  mm,
	W =  90.000 deg,	P =   0.000 deg,	R =   90.000 deg
};
P[2288]{
   GP1:
	UF : 0, UT : 6,		CONFIG : 'N U T, 0, 0, 0',
	X =  529.896  mm,	Y =   -403.102  mm,	Z =   -257.140  mm,
	W =  90.000 deg,	P =   0.000 deg,	R =   90.000 deg
};
P[2289]{
   GP1:
	UF : 0, UT : 6,		CONFIG : 'N U T, 0, 0, 0',
	X =  532.100  mm,	Y =   -401.755  mm,	Z =   -257.319  mm,
	W =  90.000 deg,	P =   0.000 deg,	R =   90.000 deg
};
P[2290]{
   GP1:
	UF : 0, UT : 6,		CONFIG : 'N U T, 0, 0, 0',
	X =  533.516  mm,	Y =   -401.076  mm,	Z =   -256.983  mm,
	W =  90.000 deg,	P =   0.000 deg,	R =   90.000 deg
};
P[2291]{
   GP1:
	UF : 0, UT : 6,		CONFIG : 'N U T, 0, 0, 0',
	X =  538.189  mm,	Y =   -397.336  mm,	Z =   -257.185  mm,
	W =  90.000 deg,	P =   0.000 deg,	R =   90.000 deg
};
P[2292]{
   GP1:
	UF : 0, UT : 6,		CONFIG : 'N U T, 0, 0, 0',
	X =  540.786  mm,	Y =   -392.834  mm,	Z =   -257.200  mm,
	W =  90.000 deg,	P =   0.000 deg,	R =   90.000 deg
};
P[2293]{
   GP1:
	UF : 0, UT : 6,		CONFIG : 'N U T, 0, 0, 0',
	X =  540.657  mm,	Y =   -383.787  mm,	Z =   -257.012  mm,
	W =  90.000 deg,	P =   0.000 deg,	R =   90.000 deg
};
P[2294]{
   GP1:
	UF : 0, UT : 6,		CONFIG : 'N U T, 0, 0, 0',
	X =  540.109  mm,	Y =   -382.659  mm,	Z =   -257.107  mm,
	W =  90.000 deg,	P =   0.000 deg,	R =   90.000 deg
};
P[2295]{
   GP1:
	UF : 0, UT : 6,		CONFIG : 'N U T, 0, 0, 0',
	X =  539.700  mm,	Y =   -381.910  mm,	Z =   -257.252  mm,
	W =  90.000 deg,	P =   0.000 deg,	R =   90.000 deg
};
P[2296]{
   GP1:
	UF : 0, UT : 6,		CONFIG : 'N U T, 0, 0, 0',
	X =  538.461  mm,	Y =   -379.433  mm,	Z =   -256.907  mm,
	W =  90.000 deg,	P =   0.000 deg,	R =   90.000 deg
};
P[2297]{
   GP1:
	UF : 0, UT : 6,		CONFIG : 'N U T, 0, 0, 0',
	X =  537.163  mm,	Y =   -377.520  mm,	Z =   -257.375  mm,
	W =  90.000 deg,	P =   0.000 deg,	R =   90.000 deg
};
P[2298]{
   GP1:
	UF : 0, UT : 6,		CONFIG : 'N U T, 0, 0, 0',
	X =  536.014  mm,	Y =   -375.195  mm,	Z =   -256.907  mm,
	W =  90.000 deg,	P =   0.000 deg,	R =   90.000 deg
};
P[2299]{
   GP1:
	UF : 0, UT : 6,		CONFIG : 'N U T, 0, 0, 0',
	X =  535.535  mm,	Y =   -374.496  mm,	Z =   -257.091  mm,
	W =  90.000 deg,	P =   0.000 deg,	R =   90.000 deg
};
P[2300]{
   GP1:
	UF : 0, UT : 6,		CONFIG : 'N U T, 0, 0, 0',
	X =  534.132  mm,	Y =   -371.921  mm,	Z =   -256.887  mm,
	W =  90.000 deg,	P =   0.000 deg,	R =   90.000 deg
};
P[2301]{
   GP1:
	UF : 0, UT : 6,		CONFIG : 'N U T, 0, 0, 0',
	X =  533.741  mm,	Y =   -371.392  mm,	Z =   -257.094  mm,
	W =  90.000 deg,	P =   0.000 deg,	R =   90.000 deg
};
P[2302]{
   GP1:
	UF : 0, UT : 6,		CONFIG : 'N U T, 0, 0, 0',
	X =  533.272  mm,	Y =   -370.602  mm,	Z =   -257.126  mm,
	W =  90.000 deg,	P =   0.000 deg,	R =   90.000 deg
};
P[2303]{
   GP1:
	UF : 0, UT : 6,		CONFIG : 'N U T, 0, 0, 0',
	X =  532.990  mm,	Y =   -369.991  mm,	Z =   -256.953  mm,
	W =  90.000 deg,	P =   0.000 deg,	R =   90.000 deg
};
P[2304]{
   GP1:
	UF : 0, UT : 6,		CONFIG : 'N U T, 0, 0, 0',
	X =  531.646  mm,	Y =   -367.761  mm,	Z =   -257.092  mm,
	W =  90.000 deg,	P =   0.000 deg,	R =   90.000 deg
};
P[2305]{
   GP1:
	UF : 0, UT : 6,		CONFIG : 'N U T, 0, 0, 0',
	X =  530.812  mm,	Y =   -366.495  mm,	Z =   -257.341  mm,
	W =  90.000 deg,	P =   0.000 deg,	R =   90.000 deg
};
P[2306]{
   GP1:
	UF : 0, UT : 6,		CONFIG : 'N U T, 0, 0, 0',
	X =  530.649  mm,	Y =   -365.902  mm,	Z =   -256.904  mm,
	W =  90.000 deg,	P =   0.000 deg,	R =   90.000 deg
};
P[2307]{
   GP1:
	UF : 0, UT : 6,		CONFIG : 'N U T, 0, 0, 0',
	X =  528.969  mm,	Y =   -363.161  mm,	Z =   -257.142  mm,
	W =  90.000 deg,	P =   0.000 deg,	R =   90.000 deg
};
P[2308]{
   GP1:
	UF : 0, UT : 6,		CONFIG : 'N U T, 0, 0, 0',
	X =  528.252  mm,	Y =   -361.890  mm,	Z =   -257.102  mm,
	W =  90.000 deg,	P =   0.000 deg,	R =   90.000 deg
};
P[2309]{
   GP1:
	UF : 0, UT : 6,		CONFIG : 'N U T, 0, 0, 0',
	X =  526.571  mm,	Y =   -359.047  mm,	Z =   -257.197  mm,
	W =  90.000 deg,	P =   0.000 deg,	R =   90.000 deg
};
P[2310]{
   GP1:
	UF : 0, UT : 6,		CONFIG : 'N U T, 0, 0, 0',
	X =  526.208  mm,	Y =   -358.255  mm,	Z =   -256.967  mm,
	W =  90.000 deg,	P =   0.000 deg,	R =   90.000 deg
};
P[2311]{
   GP1:
	UF : 0, UT : 6,		CONFIG : 'N U T, 0, 0, 0',
	X =  525.489  mm,	Y =   -357.111  mm,	Z =   -257.110  mm,
	W =  90.000 deg,	P =   0.000 deg,	R =   90.000 deg
};
P[2312]{
   GP1:
	UF : 0, UT : 6,		CONFIG : 'N U T, 0, 0, 0',
	X =  524.945  mm,	Y =   -356.078  mm,	Z =   -256.984  mm,
	W =  90.000 deg,	P =   0.000 deg,	R =   90.000 deg
};
P[2313]{
   GP1:
	UF : 0, UT : 6,		CONFIG : 'N U T, 0, 0, 0',
	X =  523.918  mm,	Y =   -354.398  mm,	Z =   -257.119  mm,
	W =  90.000 deg,	P =   0.000 deg,	R =   90.000 deg
};
P[2314]{
   GP1:
	UF : 0, UT : 6,		CONFIG : 'N U T, 0, 0, 0',
	X =  522.426  mm,	Y =   -351.848  mm,	Z =   -257.167  mm,
	W =  90.000 deg,	P =   0.000 deg,	R =   90.000 deg
};
P[2315]{
   GP1:
	UF : 0, UT : 6,		CONFIG : 'N U T, 0, 0, 0',
	X =  521.566  mm,	Y =   -350.469  mm,	Z =   -257.323  mm,
	W =  90.000 deg,	P =   0.000 deg,	R =   90.000 deg
};
P[2316]{
   GP1:
	UF : 0, UT : 6,		CONFIG : 'N U T, 0, 0, 0',
	X =  519.503  mm,	Y =   -346.845  mm,	Z =   -257.253  mm,
	W =  90.000 deg,	P =   0.000 deg,	R =   90.000 deg
};
P[2317]{
   GP1:
	UF : 0, UT : 6,		CONFIG : 'N U T, 0, 0, 0',
	X =  518.831  mm,	Y =   -345.503  mm,	Z =   -257.002  mm,
	W =  90.000 deg,	P =   0.000 deg,	R =   90.000 deg
};
P[2318]{
   GP1:
	UF : 0, UT : 6,		CONFIG : 'N U T, 0, 0, 0',
	X =  518.104  mm,	Y =   -344.425  mm,	Z =   -257.256  mm,
	W =  90.000 deg,	P =   0.000 deg,	R =   90.000 deg
};
P[2319]{
   GP1:
	UF : 0, UT : 6,		CONFIG : 'N U T, 0, 0, 0',
	X =  517.548  mm,	Y =   -343.505  mm,	Z =   -257.316  mm,
	W =  90.000 deg,	P =   0.000 deg,	R =   90.000 deg
};
P[2320]{
   GP1:
	UF : 0, UT : 6,		CONFIG : 'N U T, 0, 0, 0',
	X =  516.117  mm,	Y =   -341.041  mm,	Z =   -257.337  mm,
	W =  90.000 deg,	P =   0.000 deg,	R =   90.000 deg
};
P[2321]{
   GP1:
	UF : 0, UT : 6,		CONFIG : 'N U T, 0, 0, 0',
	X =  515.740  mm,	Y =   -340.387  mm,	Z =   -257.336  mm,
	W =  90.000 deg,	P =   0.000 deg,	R =   90.000 deg
};
P[2322]{
   GP1:
	UF : 0, UT : 6,		CONFIG : 'N U T, 0, 0, 0',
	X =  513.713  mm,	Y =   -336.769  mm,	Z =   -257.182  mm,
	W =  90.000 deg,	P =   0.000 deg,	R =   90.000 deg
};
P[2323]{
   GP1:
	UF : 0, UT : 6,		CONFIG : 'N U T, 0, 0, 0',
	X =  512.056  mm,	Y =   -333.976  mm,	Z =   -257.291  mm,
	W =  90.000 deg,	P =   0.000 deg,	R =   90.000 deg
};
P[2324]{
   GP1:
	UF : 0, UT : 6,		CONFIG : 'N U T, 0, 0, 0',
	X =  510.655  mm,	Y =   -331.529  mm,	Z =   -257.264  mm,
	W =  90.000 deg,	P =   0.000 deg,	R =   90.000 deg
};
P[2325]{
   GP1:
	UF : 0, UT : 6,		CONFIG : 'N U T, 0, 0, 0',
	X =  510.105  mm,	Y =   -330.322  mm,	Z =   -256.906  mm,
	W =  90.000 deg,	P =   0.000 deg,	R =   90.000 deg
};
P[2326]{
   GP1:
	UF : 0, UT : 6,		CONFIG : 'N U T, 0, 0, 0',
	X =  508.399  mm,	Y =   -327.445  mm,	Z =   -257.015  mm,
	W =  90.000 deg,	P =   0.000 deg,	R =   90.000 deg
};
P[2327]{
   GP1:
	UF : 0, UT : 6,		CONFIG : 'N U T, 0, 0, 0',
	X =  507.705  mm,	Y =   -326.323  mm,	Z =   -257.125  mm,
	W =  90.000 deg,	P =   0.000 deg,	R =   90.000 deg
};
P[2328]{
   GP1:
	UF : 0, UT : 6,		CONFIG : 'N U T, 0, 0, 0',
	X =  505.298  mm,	Y =   -321.993  mm,	Z =   -256.900  mm,
	W =  90.000 deg,	P =   0.000 deg,	R =   90.000 deg
};
P[2329]{
   GP1:
	UF : 0, UT : 6,		CONFIG : 'N U T, 0, 0, 0',
	X =  504.670  mm,	Y =   -321.048  mm,	Z =   -257.102  mm,
	W =  90.000 deg,	P =   0.000 deg,	R =   90.000 deg
};
P[2330]{
   GP1:
	UF : 0, UT : 6,		CONFIG : 'N U T, 0, 0, 0',
	X =  504.326  mm,	Y =   -320.300  mm,	Z =   -256.887  mm,
	W =  90.000 deg,	P =   0.000 deg,	R =   90.000 deg
};
P[2331]{
   GP1:
	UF : 0, UT : 6,		CONFIG : 'N U T, 0, 0, 0',
	X =  501.930  mm,	Y =   -316.275  mm,	Z =   -257.063  mm,
	W =  90.000 deg,	P =   0.000 deg,	R =   90.000 deg
};
P[2332]{
   GP1:
	UF : 0, UT : 6,		CONFIG : 'N U T, 0, 0, 0',
	X =  501.384  mm,	Y =   -315.473  mm,	Z =   -257.263  mm,
	W =  90.000 deg,	P =   0.000 deg,	R =   90.000 deg
};
P[2333]{
   GP1:
	UF : 0, UT : 6,		CONFIG : 'N U T, 0, 0, 0',
	X =  499.114  mm,	Y =   -311.406  mm,	Z =   -257.074  mm,
	W =  90.000 deg,	P =   0.000 deg,	R =   90.000 deg
};
P[2334]{
   GP1:
	UF : 0, UT : 6,		CONFIG : 'N U T, 0, 0, 0',
	X =  498.617  mm,	Y =   -310.578  mm,	Z =   -257.119  mm,
	W =  90.000 deg,	P =   0.000 deg,	R =   90.000 deg
};
P[2335]{
   GP1:
	UF : 0, UT : 6,		CONFIG : 'N U T, 0, 0, 0',
	X =  497.584  mm,	Y =   -308.771  mm,	Z =   -257.094  mm,
	W =  90.000 deg,	P =   0.000 deg,	R =   90.000 deg
};
P[2336]{
   GP1:
	UF : 0, UT : 6,		CONFIG : 'N U T, 0, 0, 0',
	X =  496.565  mm,	Y =   -307.021  mm,	Z =   -257.115  mm,
	W =  90.000 deg,	P =   0.000 deg,	R =   90.000 deg
};
P[2337]{
   GP1:
	UF : 0, UT : 6,		CONFIG : 'N U T, 0, 0, 0',
	X =  494.797  mm,	Y =   -303.981  mm,	Z =   -257.147  mm,
	W =  90.000 deg,	P =   0.000 deg,	R =   90.000 deg
};
P[2338]{
   GP1:
	UF : 0, UT : 6,		CONFIG : 'N U T, 0, 0, 0',
	X =  494.119  mm,	Y =   -302.697  mm,	Z =   -256.992  mm,
	W =  90.000 deg,	P =   0.000 deg,	R =   90.000 deg
};
P[2339]{
   GP1:
	UF : 0, UT : 6,		CONFIG : 'N U T, 0, 0, 0',
	X =  493.316  mm,	Y =   -301.556  mm,	Z =   -257.343  mm,
	W =  90.000 deg,	P =   0.000 deg,	R =   90.000 deg
};
P[2340]{
   GP1:
	UF : 0, UT : 6,		CONFIG : 'N U T, 0, 0, 0',
	X =  492.952  mm,	Y =   -300.705  mm,	Z =   -257.033  mm,
	W =  90.000 deg,	P =   0.000 deg,	R =   90.000 deg
};
P[2341]{
   GP1:
	UF : 0, UT : 6,		CONFIG : 'N U T, 0, 0, 0',
	X =  491.685  mm,	Y =   -298.702  mm,	Z =   -257.302  mm,
	W =  90.000 deg,	P =   0.000 deg,	R =   90.000 deg
};
P[2342]{
   GP1:
	UF : 0, UT : 6,		CONFIG : 'N U T, 0, 0, 0',
	X =  491.046  mm,	Y =   -297.561  mm,	Z =   -257.253  mm,
	W =  90.000 deg,	P =   0.000 deg,	R =   90.000 deg
};
P[2343]{
   GP1:
	UF : 0, UT : 6,		CONFIG : 'N U T, 0, 0, 0',
	X =  490.573  mm,	Y =   -296.503  mm,	Z =   -256.919  mm,
	W =  90.000 deg,	P =   0.000 deg,	R =   90.000 deg
};
P[2344]{
   GP1:
	UF : 0, UT : 6,		CONFIG : 'N U T, 0, 0, 0',
	X =  489.795  mm,	Y =   -295.462  mm,	Z =   -257.346  mm,
	W =  90.000 deg,	P =   0.000 deg,	R =   90.000 deg
};
P[2345]{
   GP1:
	UF : 0, UT : 6,		CONFIG : 'N U T, 0, 0, 0',
	X =  489.193  mm,	Y =   -294.248  mm,	Z =   -257.106  mm,
	W =  90.000 deg,	P =   0.000 deg,	R =   90.000 deg
};
P[2346]{
   GP1:
	UF : 0, UT : 6,		CONFIG : 'N U T, 0, 0, 0',
	X =  488.672  mm,	Y =   -293.425  mm,	Z =   -257.218  mm,
	W =  90.000 deg,	P =   0.000 deg,	R =   90.000 deg
};
P[2347]{
   GP1:
	UF : 0, UT : 6,		CONFIG : 'N U T, 0, 0, 0',
	X =  487.228  mm,	Y =   -290.702  mm,	Z =   -256.909  mm,
	W =  90.000 deg,	P =   0.000 deg,	R =   90.000 deg
};
P[2348]{
   GP1:
	UF : 0, UT : 6,		CONFIG : 'N U T, 0, 0, 0',
	X =  485.347  mm,	Y =   -287.724  mm,	Z =   -257.299  mm,
	W =  90.000 deg,	P =   0.000 deg,	R =   90.000 deg
};
P[2349]{
   GP1:
	UF : 0, UT : 6,		CONFIG : 'N U T, 0, 0, 0',
	X =  484.866  mm,	Y =   -286.838  mm,	Z =   -257.225  mm,
	W =  90.000 deg,	P =   0.000 deg,	R =   90.000 deg
};
P[2350]{
   GP1:
	UF : 0, UT : 6,		CONFIG : 'N U T, 0, 0, 0',
	X =  483.693  mm,	Y =   -284.823  mm,	Z =   -257.249  mm,
	W =  90.000 deg,	P =   0.000 deg,	R =   90.000 deg
};
P[2351]{
   GP1:
	UF : 0, UT : 6,		CONFIG : 'N U T, 0, 0, 0',
	X =  482.380  mm,	Y =   -282.501  mm,	Z =   -257.183  mm,
	W =  90.000 deg,	P =   0.000 deg,	R =   90.000 deg
};
P[2352]{
   GP1:
	UF : 0, UT : 6,		CONFIG : 'N U T, 0, 0, 0',
	X =  478.139  mm,	Y =   -275.232  mm,	Z =   -257.290  mm,
	W =  90.000 deg,	P =   0.000 deg,	R =   90.000 deg
};
P[2353]{
   GP1:
	UF : 0, UT : 6,		CONFIG : 'N U T, 0, 0, 0',
	X =  476.944  mm,	Y =   -273.123  mm,	Z =   -257.234  mm,
	W =  90.000 deg,	P =   0.000 deg,	R =   90.000 deg
};
P[2354]{
   GP1:
	UF : 0, UT : 6,		CONFIG : 'N U T, 0, 0, 0',
	X =  474.569  mm,	Y =   -269.061  mm,	Z =   -257.304  mm,
	W =  90.000 deg,	P =   0.000 deg,	R =   90.000 deg
};
P[2355]{
   GP1:
	UF : 0, UT : 6,		CONFIG : 'N U T, 0, 0, 0',
	X =  473.242  mm,	Y =   -266.713  mm,	Z =   -257.237  mm,
	W =  90.000 deg,	P =   0.000 deg,	R =   90.000 deg
};
P[2356]{
   GP1:
	UF : 0, UT : 6,		CONFIG : 'N U T, 0, 0, 0',
	X =  472.767  mm,	Y =   -265.851  mm,	Z =   -257.180  mm,
	W =  90.000 deg,	P =   0.000 deg,	R =   90.000 deg
};
P[2357]{
   GP1:
	UF : 0, UT : 6,		CONFIG : 'N U T, 0, 0, 0',
	X =  471.514  mm,	Y =   -263.800  mm,	Z =   -257.345  mm,
	W =  90.000 deg,	P =   0.000 deg,	R =   90.000 deg
};
P[2358]{
   GP1:
	UF : 0, UT : 6,		CONFIG : 'N U T, 0, 0, 0',
	X =  470.452  mm,	Y =   -261.841  mm,	Z =   -257.180  mm,
	W =  90.000 deg,	P =   0.000 deg,	R =   90.000 deg
};
P[2359]{
   GP1:
	UF : 0, UT : 6,		CONFIG : 'N U T, 0, 0, 0',
	X =  468.945  mm,	Y =   -259.284  mm,	Z =   -257.252  mm,
	W =  90.000 deg,	P =   0.000 deg,	R =   90.000 deg
};
P[2360]{
   GP1:
	UF : 0, UT : 6,		CONFIG : 'N U T, 0, 0, 0',
	X =  468.336  mm,	Y =   -258.191  mm,	Z =   -257.200  mm,
	W =  90.000 deg,	P =   0.000 deg,	R =   90.000 deg
};
P[2361]{
   GP1:
	UF : 0, UT : 6,		CONFIG : 'N U T, 0, 0, 0',
	X =  466.909  mm,	Y =   -255.780  mm,	Z =   -257.285  mm,
	W =  90.000 deg,	P =   0.000 deg,	R =   90.000 deg
};
P[2362]{
   GP1:
	UF : 0, UT : 6,		CONFIG : 'N U T, 0, 0, 0',
	X =  466.301  mm,	Y =   -254.602  mm,	Z =   -257.110  mm,
	W =  90.000 deg,	P =   0.000 deg,	R =   90.000 deg
};
P[2363]{
   GP1:
	UF : 0, UT : 6,		CONFIG : 'N U T, 0, 0, 0',
	X =  465.675  mm,	Y =   -253.637  mm,	Z =   -257.277  mm,
	W =  90.000 deg,	P =   0.000 deg,	R =   90.000 deg
};
P[2364]{
   GP1:
	UF : 0, UT : 6,		CONFIG : 'N U T, 0, 0, 0',
	X =  462.511  mm,	Y =   -247.907  mm,	Z =   -256.926  mm,
	W =  90.000 deg,	P =   0.000 deg,	R =   90.000 deg
};
P[2365]{
   GP1:
	UF : 0, UT : 6,		CONFIG : 'N U T, 0, 0, 0',
	X =  461.673  mm,	Y =   -246.438  mm,	Z =   -256.901  mm,
	W =  90.000 deg,	P =   0.000 deg,	R =   90.000 deg
};
P[2366]{
   GP1:
	UF : 0, UT : 6,		CONFIG : 'N U T, 0, 0, 0',
	X =  461.075  mm,	Y =   -245.671  mm,	Z =   -257.278  mm,
	W =  90.000 deg,	P =   0.000 deg,	R =   90.000 deg
};
P[2367]{
   GP1:
	UF : 0, UT : 6,		CONFIG : 'N U T, 0, 0, 0',
	X =  460.596  mm,	Y =   -244.837  mm,	Z =   -257.272  mm,
	W =  90.000 deg,	P =   0.000 deg,	R =   90.000 deg
};
P[2368]{
   GP1:
	UF : 0, UT : 6,		CONFIG : 'N U T, 0, 0, 0',
	X =  459.248  mm,	Y =   -242.232  mm,	Z =   -256.892  mm,
	W =  90.000 deg,	P =   0.000 deg,	R =   90.000 deg
};
P[2369]{
   GP1:
	UF : 0, UT : 6,		CONFIG : 'N U T, 0, 0, 0',
	X =  458.694  mm,	Y =   -241.618  mm,	Z =   -257.375  mm,
	W =  90.000 deg,	P =   0.000 deg,	R =   90.000 deg
};
P[2370]{
   GP1:
	UF : 0, UT : 6,		CONFIG : 'N U T, 0, 0, 0',
	X =  458.562  mm,	Y =   -241.084  mm,	Z =   -256.947  mm,
	W =  90.000 deg,	P =   0.000 deg,	R =   90.000 deg
};
P[2371]{
   GP1:
	UF : 0, UT : 6,		CONFIG : 'N U T, 0, 0, 0',
	X =  456.368  mm,	Y =   -237.447  mm,	Z =   -257.179  mm,
	W =  90.000 deg,	P =   0.000 deg,	R =   90.000 deg
};
P[2372]{
   GP1:
	UF : 0, UT : 6,		CONFIG : 'N U T, 0, 0, 0',
	X =  455.822  mm,	Y =   -236.628  mm,	Z =   -257.353  mm,
	W =  90.000 deg,	P =   0.000 deg,	R =   90.000 deg
};
P[2373]{
   GP1:
	UF : 0, UT : 6,		CONFIG : 'N U T, 0, 0, 0',
	X =  455.496  mm,	Y =   -235.871  mm,	Z =   -257.085  mm,
	W =  90.000 deg,	P =   0.000 deg,	R =   90.000 deg
};
P[2374]{
   GP1:
	UF : 0, UT : 6,		CONFIG : 'N U T, 0, 0, 0',
	X =  454.962  mm,	Y =   -235.155  mm,	Z =   -257.379  mm,
	W =  90.000 deg,	P =   0.000 deg,	R =   90.000 deg
};
P[2375]{
   GP1:
	UF : 0, UT : 6,		CONFIG : 'N U T, 0, 0, 0',
	X =  452.041  mm,	Y =   -229.977  mm,	Z =   -257.210  mm,
	W =  90.000 deg,	P =   0.000 deg,	R =   90.000 deg
};
P[2376]{
   GP1:
	UF : 0, UT : 6,		CONFIG : 'N U T, 0, 0, 0',
	X =  451.366  mm,	Y =   -228.921  mm,	Z =   -257.372  mm,
	W =  90.000 deg,	P =   0.000 deg,	R =   90.000 deg
};
P[2377]{
   GP1:
	UF : 0, UT : 6,		CONFIG : 'N U T, 0, 0, 0',
	X =  450.930  mm,	Y =   -228.107  mm,	Z =   -257.285  mm,
	W =  90.000 deg,	P =   0.000 deg,	R =   90.000 deg
};
P[2378]{
   GP1:
	UF : 0, UT : 6,		CONFIG : 'N U T, 0, 0, 0',
	X =  450.253  mm,	Y =   -226.728  mm,	Z =   -256.997  mm,
	W =  90.000 deg,	P =   0.000 deg,	R =   90.000 deg
};
P[2379]{
   GP1:
	UF : 0, UT : 6,		CONFIG : 'N U T, 0, 0, 0',
	X =  448.995  mm,	Y =   -224.677  mm,	Z =   -257.175  mm,
	W =  90.000 deg,	P =   0.000 deg,	R =   90.000 deg
};
P[2380]{
   GP1:
	UF : 0, UT : 6,		CONFIG : 'N U T, 0, 0, 0',
	X =  447.424  mm,	Y =   -221.757  mm,	Z =   -256.899  mm,
	W =  90.000 deg,	P =   0.000 deg,	R =   90.000 deg
};
P[2381]{
   GP1:
	UF : 0, UT : 6,		CONFIG : 'N U T, 0, 0, 0',
	X =  444.671  mm,	Y =   -217.047  mm,	Z =   -256.978  mm,
	W =  90.000 deg,	P =   0.000 deg,	R =   90.000 deg
};
P[2382]{
   GP1:
	UF : 0, UT : 6,		CONFIG : 'N U T, 0, 0, 0',
	X =  443.849  mm,	Y =   -215.891  mm,	Z =   -257.353  mm,
	W =  90.000 deg,	P =   0.000 deg,	R =   90.000 deg
};
P[2383]{
   GP1:
	UF : 0, UT : 6,		CONFIG : 'N U T, 0, 0, 0',
	X =  443.198  mm,	Y =   -214.636  mm,	Z =   -257.174  mm,
	W =  90.000 deg,	P =   0.000 deg,	R =   90.000 deg
};
P[2384]{
   GP1:
	UF : 0, UT : 6,		CONFIG : 'N U T, 0, 0, 0',
	X =  441.373  mm,	Y =   -211.561  mm,	Z =   -257.295  mm,
	W =  90.000 deg,	P =   0.000 deg,	R =   90.000 deg
};
P[2385]{
   GP1:
	UF : 0, UT : 6,		CONFIG : 'N U T, 0, 0, 0',
	X =  440.315  mm,	Y =   -209.465  mm,	Z =   -256.925  mm,
	W =  90.000 deg,	P =   0.000 deg,	R =   90.000 deg
};
P[2386]{
   GP1:
	UF : 0, UT : 6,		CONFIG : 'N U T, 0, 0, 0',
	X =  439.413  mm,	Y =   -208.120  mm,	Z =   -257.231  mm,
	W =  90.000 deg,	P =   0.000 deg,	R =   90.000 deg
};
P[2387]{
   GP1:
	UF : 0, UT : 6,		CONFIG : 'N U T, 0, 0, 0',
	X =  438.533  mm,	Y =   -206.506  mm,	Z =   -257.105  mm,
	W =  90.000 deg,	P =   0.000 deg,	R =   90.000 deg
};
P[2388]{
   GP1:
	UF : 0, UT : 6,		CONFIG : 'N U T, 0, 0, 0',
	X =  437.236  mm,	Y =   -204.270  mm,	Z =   -257.117  mm,
	W =  90.000 deg,	P =   0.000 deg,	R =   90.000 deg
};
P[2389]{
   GP1:
	UF : 0, UT : 6,		CONFIG : 'N U T, 0, 0, 0',
	X =  434.654  mm,	Y =   -199.838  mm,	Z =   -257.176  mm,
	W =  90.000 deg,	P =   0.000 deg,	R =   90.000 deg
};
P[2390]{
   GP1:
	UF : 0, UT : 6,		CONFIG : 'N U T, 0, 0, 0',
	X =  433.527  mm,	Y =   -197.974  mm,	Z =   -257.298  mm,
	W =  90.000 deg,	P =   0.000 deg,	R =   90.000 deg
};
P[2391]{
   GP1:
	UF : 0, UT : 6,		CONFIG : 'N U T, 0, 0, 0',
	X =  433.182  mm,	Y =   -197.092  mm,	Z =   -256.898  mm,
	W =  90.000 deg,	P =   0.000 deg,	R =   90.000 deg
};
P[2392]{
   GP1:
	UF : 0, UT : 6,		CONFIG : 'N U T, 0, 0, 0',
	X =  431.419  mm,	Y =   -194.347  mm,	Z =   -257.330  mm,
	W =  90.000 deg,	P =   0.000 deg,	R =   90.000 deg
};
P[2393]{
   GP1:
	UF : 0, UT : 6,		CONFIG : 'N U T, 0, 0, 0',
	X =  428.412  mm,	Y =   -189.010  mm,	Z =   -257.151  mm,
	W =  90.000 deg,	P =   0.000 deg,	R =   90.000 deg
};
P[2394]{
   GP1:
	UF : 0, UT : 6,		CONFIG : 'N U T, 0, 0, 0',
	X =  426.302  mm,	Y =   -185.419  mm,	Z =   -257.240  mm,
	W =  90.000 deg,	P =   0.000 deg,	R =   90.000 deg
};
P[2395]{
   GP1:
	UF : 0, UT : 6,		CONFIG : 'N U T, 0, 0, 0',
	X =  425.712  mm,	Y =   -184.255  mm,	Z =   -257.040  mm,
	W =  90.000 deg,	P =   0.000 deg,	R =   90.000 deg
};
P[2396]{
   GP1:
	UF : 0, UT : 6,		CONFIG : 'N U T, 0, 0, 0',
	X =  425.074  mm,	Y =   -183.268  mm,	Z =   -257.206  mm,
	W =  90.000 deg,	P =   0.000 deg,	R =   90.000 deg
};
P[2397]{
   GP1:
	UF : 0, UT : 6,		CONFIG : 'N U T, 0, 0, 0',
	X =  424.057  mm,	Y =   -181.460  mm,	Z =   -257.140  mm,
	W =  90.000 deg,	P =   0.000 deg,	R =   90.000 deg
};
P[2398]{
   GP1:
	UF : 0, UT : 6,		CONFIG : 'N U T, 0, 0, 0',
	X =  422.877  mm,	Y =   -179.526  mm,	Z =   -257.295  mm,
	W =  90.000 deg,	P =   0.000 deg,	R =   90.000 deg
};
P[2399]{
   GP1:
	UF : 0, UT : 6,		CONFIG : 'N U T, 0, 0, 0',
	X =  421.464  mm,	Y =   -176.948  mm,	Z =   -257.110  mm,
	W =  90.000 deg,	P =   0.000 deg,	R =   90.000 deg
};
P[2400]{
   GP1:
	UF : 0, UT : 6,		CONFIG : 'N U T, 0, 0, 0',
	X =  419.906  mm,	Y =   -174.428  mm,	Z =   -257.361  mm,
	W =  90.000 deg,	P =   0.000 deg,	R =   90.000 deg
};
P[2401]{
   GP1:
	UF : 0, UT : 6,		CONFIG : 'N U T, 0, 0, 0',
	X =  418.982  mm,	Y =   -172.625  mm,	Z =   -257.075  mm,
	W =  90.000 deg,	P =   0.000 deg,	R =   90.000 deg
};
P[2402]{
   GP1:
	UF : 0, UT : 6,		CONFIG : 'N U T, 0, 0, 0',
	X =  413.838  mm,	Y =   -163.889  mm,	Z =   -257.318  mm,
	W =  90.000 deg,	P =   0.000 deg,	R =   90.000 deg
};
P[2403]{
   GP1:
	UF : 0, UT : 6,		CONFIG : 'N U T, 0, 0, 0',
	X =  412.944  mm,	Y =   -162.338  mm,	Z =   -257.313  mm,
	W =  90.000 deg,	P =   0.000 deg,	R =   90.000 deg
};
P[2404]{
   GP1:
	UF : 0, UT : 6,		CONFIG : 'N U T, 0, 0, 0',
	X =  411.427  mm,	Y =   -159.589  mm,	Z =   -257.145  mm,
	W =  90.000 deg,	P =   0.000 deg,	R =   90.000 deg
};
P[2405]{
   GP1:
	UF : 0, UT : 6,		CONFIG : 'N U T, 0, 0, 0',
	X =  410.866  mm,	Y =   -158.571  mm,	Z =   -257.078  mm,
	W =  90.000 deg,	P =   0.000 deg,	R =   90.000 deg
};
P[2406]{
   GP1:
	UF : 0, UT : 6,		CONFIG : 'N U T, 0, 0, 0',
	X =  409.828  mm,	Y =   -156.769  mm,	Z =   -257.075  mm,
	W =  90.000 deg,	P =   0.000 deg,	R =   90.000 deg
};
P[2407]{
   GP1:
	UF : 0, UT : 6,		CONFIG : 'N U T, 0, 0, 0',
	X =  407.816  mm,	Y =   -153.213  mm,	Z =   -256.973  mm,
	W =  90.000 deg,	P =   0.000 deg,	R =   90.000 deg
};
P[2408]{
   GP1:
	UF : 0, UT : 6,		CONFIG : 'N U T, 0, 0, 0',
	X =  404.657  mm,	Y =   -147.872  mm,	Z =   -257.158  mm,
	W =  90.000 deg,	P =   0.000 deg,	R =   90.000 deg
};
P[2409]{
   GP1:
	UF : 0, UT : 6,		CONFIG : 'N U T, 0, 0, 0',
	X =  403.707  mm,	Y =   -146.037  mm,	Z =   -256.889  mm,
	W =  90.000 deg,	P =   0.000 deg,	R =   90.000 deg
};
P[2410]{
   GP1:
	UF : 0, UT : 6,		CONFIG : 'N U T, 0, 0, 0',
	X =  402.311  mm,	Y =   -143.764  mm,	Z =   -257.095  mm,
	W =  90.000 deg,	P =   0.000 deg,	R =   90.000 deg
};
P[2411]{
   GP1:
	UF : 0, UT : 6,		CONFIG : 'N U T, 0, 0, 0',
	X =  399.702  mm,	Y =   -139.381  mm,	Z =   -257.282  mm,
	W =  90.000 deg,	P =   0.000 deg,	R =   90.000 deg
};
P[2412]{
   GP1:
	UF : 0, UT : 6,		CONFIG : 'N U T, 0, 0, 0',
	X =  399.296  mm,	Y =   -138.622  mm,	Z =   -257.207  mm,
	W =  90.000 deg,	P =   0.000 deg,	R =   90.000 deg
};
P[2413]{
   GP1:
	UF : 0, UT : 6,		CONFIG : 'N U T, 0, 0, 0',
	X =  398.752  mm,	Y =   -137.767  mm,	Z =   -257.326  mm,
	W =  90.000 deg,	P =   0.000 deg,	R =   90.000 deg
};
P[2414]{
   GP1:
	UF : 0, UT : 6,		CONFIG : 'N U T, 0, 0, 0',
	X =  395.866  mm,	Y =   -132.749  mm,	Z =   -257.300  mm,
	W =  90.000 deg,	P =   0.000 deg,	R =   90.000 deg
};
P[2415]{
   GP1:
	UF : 0, UT : 6,		CONFIG : 'N U T, 0, 0, 0',
	X =  392.409  mm,	Y =   -126.701  mm,	Z =   -257.214  mm,
	W =  90.000 deg,	P =   0.000 deg,	R =   90.000 deg
};
P[2416]{
   GP1:
	UF : 0, UT : 6,		CONFIG : 'N U T, 0, 0, 0',
	X =  389.971  mm,	Y =   -122.493  mm,	Z =   -257.236  mm,
	W =  90.000 deg,	P =   0.000 deg,	R =   90.000 deg
};
P[2417]{
   GP1:
	UF : 0, UT : 6,		CONFIG : 'N U T, 0, 0, 0',
	X =  388.275  mm,	Y =   -119.514  mm,	Z =   -257.176  mm,
	W =  90.000 deg,	P =   0.000 deg,	R =   90.000 deg
};
P[2418]{
   GP1:
	UF : 0, UT : 6,		CONFIG : 'N U T, 0, 0, 0',
	X =  387.493  mm,	Y =   -117.966  mm,	Z =   -256.903  mm,
	W =  90.000 deg,	P =   0.000 deg,	R =   90.000 deg
};
P[2419]{
   GP1:
	UF : 0, UT : 6,		CONFIG : 'N U T, 0, 0, 0',
	X =  386.671  mm,	Y =   -116.834  mm,	Z =   -257.312  mm,
	W =  90.000 deg,	P =   0.000 deg,	R =   90.000 deg
};
P[2420]{
   GP1:
	UF : 0, UT : 6,		CONFIG : 'N U T, 0, 0, 0',
	X =  386.217  mm,	Y =   -116.067  mm,	Z =   -257.340  mm,
	W =  90.000 deg,	P =   0.000 deg,	R =   90.000 deg
};
P[2421]{
   GP1:
	UF : 0, UT : 6,		CONFIG : 'N U T, 0, 0, 0',
	X =  385.776  mm,	Y =   -115.185  mm,	Z =   -257.177  mm,
	W =  90.000 deg,	P =   0.000 deg,	R =   90.000 deg
};
P[2422]{
   GP1:
	UF : 0, UT : 6,		CONFIG : 'N U T, 0, 0, 0',
	X =  384.503  mm,	Y =   -113.020  mm,	Z =   -257.230  mm,
	W =  90.000 deg,	P =   0.000 deg,	R =   90.000 deg
};
P[2423]{
   GP1:
	UF : 0, UT : 6,		CONFIG : 'N U T, 0, 0, 0',
	X =  383.638  mm,	Y =   -111.346  mm,	Z =   -256.985  mm,
	W =  90.000 deg,	P =   0.000 deg,	R =   90.000 deg
};
P[2424]{
   GP1:
	UF : 0, UT : 6,		CONFIG : 'N U T, 0, 0, 0',
	X =  381.205  mm,	Y =   -107.407  mm,	Z =   -257.371  mm,
	W =  90.000 deg,	P =   0.000 deg,	R =   90.000 deg
};
P[2425]{
   GP1:
	UF : 0, UT : 6,		CONFIG : 'N U T, 0, 0, 0',
	X =  380.745  mm,	Y =   -106.523  mm,	Z =   -257.246  mm,
	W =  90.000 deg,	P =   0.000 deg,	R =   90.000 deg
};
P[2426]{
   GP1:
	UF : 0, UT : 6,		CONFIG : 'N U T, 0, 0, 0',
	X =  379.150  mm,	Y =   -103.854  mm,	Z =   -257.379  mm,
	W =  90.000 deg,	P =   0.000 deg,	R =   90.000 deg
};
P[2427]{
   GP1:
	UF : 0, UT : 6,		CONFIG : 'N U T, 0, 0, 0',
	X =  376.279  mm,	Y =   -98.867  mm,	Z =   -257.358  mm,
	W =  90.000 deg,	P =   0.000 deg,	R =   90.000 deg
};
P[2428]{
   GP1:
	UF : 0, UT : 6,		CONFIG : 'N U T, 0, 0, 0',
	X =  375.164  mm,	Y =   -96.751  mm,	Z =   -257.100  mm,
	W =  90.000 deg,	P =   0.000 deg,	R =   90.000 deg
};
P[2429]{
   GP1:
	UF : 0, UT : 6,		CONFIG : 'N U T, 0, 0, 0',
	X =  374.741  mm,	Y =   -95.894  mm,	Z =   -256.924  mm,
	W =  90.000 deg,	P =   0.000 deg,	R =   90.000 deg
};
P[2430]{
   GP1:
	UF : 0, UT : 6,		CONFIG : 'N U T, 0, 0, 0',
	X =  374.264  mm,	Y =   -95.362  mm,	Z =   -257.336  mm,
	W =  90.000 deg,	P =   0.000 deg,	R =   90.000 deg
};
P[2431]{
   GP1:
	UF : 0, UT : 6,		CONFIG : 'N U T, 0, 0, 0',
	X =  373.767  mm,	Y =   -94.206  mm,	Z =   -256.925  mm,
	W =  90.000 deg,	P =   0.000 deg,	R =   90.000 deg
};
P[2432]{
   GP1:
	UF : 0, UT : 6,		CONFIG : 'N U T, 0, 0, 0',
	X =  371.711  mm,	Y =   -90.784  mm,	Z =   -257.118  mm,
	W =  90.000 deg,	P =   0.000 deg,	R =   90.000 deg
};
P[2433]{
   GP1:
	UF : 0, UT : 6,		CONFIG : 'N U T, 0, 0, 0',
	X =  370.868  mm,	Y =   -89.513  mm,	Z =   -257.381  mm,
	W =  90.000 deg,	P =   0.000 deg,	R =   90.000 deg
};
P[2434]{
   GP1:
	UF : 0, UT : 6,		CONFIG : 'N U T, 0, 0, 0',
	X =  368.188  mm,	Y =   -84.945  mm,	Z =   -257.066  mm,
	W =  90.000 deg,	P =   0.000 deg,	R =   90.000 deg
};
P[2435]{
   GP1:
	UF : 0, UT : 6,		CONFIG : 'N U T, 0, 0, 0',
	X =  366.575  mm,	Y =   -82.960  mm,	Z =   -256.889  mm,
	W =  90.000 deg,	P =   0.000 deg,	R =   90.000 deg
};
P[2436]{
   GP1:
	UF : 0, UT : 6,		CONFIG : 'N U T, 0, 0, 0',
	X =  365.981  mm,	Y =   -82.434  mm,	Z =   -256.919  mm,
	W =  90.000 deg,	P =   0.000 deg,	R =   90.000 deg
};
P[2437]{
   GP1:
	UF : 0, UT : 6,		CONFIG : 'N U T, 0, 0, 0',
	X =  364.938  mm,	Y =   -81.796  mm,	Z =   -257.267  mm,
	W =  90.000 deg,	P =   0.000 deg,	R =   90.000 deg
};
P[2438]{
   GP1:
	UF : 0, UT : 6,		CONFIG : 'N U T, 0, 0, 0',
	X =  363.991  mm,	Y =   -81.126  mm,	Z =   -257.123  mm,
	W =  90.000 deg,	P =   0.000 deg,	R =   90.000 deg
};
P[2439]{
   GP1:
	UF : 0, UT : 6,		CONFIG : 'N U T, 0, 0, 0',
	X =  362.743  mm,	Y =   -80.542  mm,	Z =   -257.284  mm,
	W =  90.000 deg,	P =   0.000 deg,	R =   90.000 deg
};
P[2440]{
   GP1:
	UF : 0, UT : 6,		CONFIG : 'N U T, 0, 0, 0',
	X =  359.288  mm,	Y =   -79.583  mm,	Z =   -257.382  mm,
	W =  90.000 deg,	P =   0.000 deg,	R =   90.000 deg
};
P[2441]{
   GP1:
	UF : 0, UT : 6,		CONFIG : 'N U T, 0, 0, 0',
	X =  358.306  mm,	Y =   -79.342  mm,	Z =   -257.136  mm,
	W =  90.000 deg,	P =   0.000 deg,	R =   90.000 deg
};
P[2442]{
   GP1:
	UF : 0, UT : 6,		CONFIG : 'N U T, 0, 0, 0',
	X =  357.224  mm,	Y =   -79.391  mm,	Z =   -257.272  mm,
	W =  90.000 deg,	P =   0.000 deg,	R =   90.000 deg
};
P[2443]{
   GP1:
	UF : 0, UT : 6,		CONFIG : 'N U T, 0, 0, 0',
	X =  355.298  mm,	Y =   -79.527  mm,	Z =   -257.266  mm,
	W =  90.000 deg,	P =   0.000 deg,	R =   90.000 deg
};
P[2444]{
   GP1:
	UF : 0, UT : 6,		CONFIG : 'N U T, 0, 0, 0',
	X =  352.448  mm,	Y =   -80.270  mm,	Z =   -257.255  mm,
	W =  90.000 deg,	P =   0.000 deg,	R =   90.000 deg
};
P[2445]{
   GP1:
	UF : 0, UT : 6,		CONFIG : 'N U T, 0, 0, 0',
	X =  351.767  mm,	Y =   -80.426  mm,	Z =   -256.918  mm,
	W =  90.000 deg,	P =   0.000 deg,	R =   90.000 deg
};
P[2446]{
   GP1:
	UF : 0, UT : 6,		CONFIG : 'N U T, 0, 0, 0',
	X =  350.548  mm,	Y =   -81.136  mm,	Z =   -257.263  mm,
	W =  90.000 deg,	P =   0.000 deg,	R =   90.000 deg
};
P[2447]{
   GP1:
	UF : 0, UT : 6,		CONFIG : 'N U T, 0, 0, 0',
	X =  348.946  mm,	Y =   -81.937  mm,	Z =   -257.070  mm,
	W =  90.000 deg,	P =   0.000 deg,	R =   90.000 deg
};
P[2448]{
   GP1:
	UF : 0, UT : 6,		CONFIG : 'N U T, 0, 0, 0',
	X =  347.979  mm,	Y =   -82.584  mm,	Z =   -257.281  mm,
	W =  90.000 deg,	P =   0.000 deg,	R =   90.000 deg
};
P[2449]{
   GP1:
	UF : 0, UT : 6,		CONFIG : 'N U T, 0, 0, 0',
	X =  345.242  mm,	Y =   -84.206  mm,	Z =   -257.385  mm,
	W =  90.000 deg,	P =   0.000 deg,	R =   90.000 deg
};
P[2450]{
   GP1:
	UF : 0, UT : 6,		CONFIG : 'N U T, 0, 0, 0',
	X =  340.927  mm,	Y =   -86.586  mm,	Z =   -257.114  mm,
	W =  90.000 deg,	P =   0.000 deg,	R =   90.000 deg
};
P[2451]{
   GP1:
	UF : 0, UT : 6,		CONFIG : 'N U T, 0, 0, 0',
	X =  340.100  mm,	Y =   -87.063  mm,	Z =   -257.114  mm,
	W =  90.000 deg,	P =   0.000 deg,	R =   90.000 deg
};
P[2452]{
   GP1:
	UF : 0, UT : 6,		CONFIG : 'N U T, 0, 0, 0',
	X =  336.438  mm,	Y =   -89.140  mm,	Z =   -257.024  mm,
	W =  90.000 deg,	P =   0.000 deg,	R =   90.000 deg
};
P[2453]{
   GP1:
	UF : 0, UT : 6,		CONFIG : 'N U T, 0, 0, 0',
	X =  333.802  mm,	Y =   -90.797  mm,	Z =   -257.348  mm,
	W =  90.000 deg,	P =   0.000 deg,	R =   90.000 deg
};
P[2454]{
   GP1:
	UF : 0, UT : 6,		CONFIG : 'N U T, 0, 0, 0',
	X =  330.382  mm,	Y =   -92.677  mm,	Z =   -257.119  mm,
	W =  90.000 deg,	P =   0.000 deg,	R =   90.000 deg
};
P[2455]{
   GP1:
	UF : 0, UT : 6,		CONFIG : 'N U T, 0, 0, 0',
	X =  329.044  mm,	Y =   -93.543  mm,	Z =   -257.346  mm,
	W =  90.000 deg,	P =   0.000 deg,	R =   90.000 deg
};
P[2456]{
   GP1:
	UF : 0, UT : 6,		CONFIG : 'N U T, 0, 0, 0',
	X =  328.417  mm,	Y =   -93.917  mm,	Z =   -257.376  mm,
	W =  90.000 deg,	P =   0.000 deg,	R =   90.000 deg
};
P[2457]{
   GP1:
	UF : 0, UT : 6,		CONFIG : 'N U T, 0, 0, 0',
	X =  325.933  mm,	Y =   -95.286  mm,	Z =   -257.216  mm,
	W =  90.000 deg,	P =   0.000 deg,	R =   90.000 deg
};
P[2458]{
   GP1:
	UF : 0, UT : 6,		CONFIG : 'N U T, 0, 0, 0',
	X =  324.377  mm,	Y =   -96.142  mm,	Z =   -257.112  mm,
	W =  90.000 deg,	P =   0.000 deg,	R =   90.000 deg
};
P[2459]{
   GP1:
	UF : 0, UT : 6,		CONFIG : 'N U T, 0, 0, 0',
	X =  321.926  mm,	Y =   -97.473  mm,	Z =   -256.910  mm,
	W =  90.000 deg,	P =   0.000 deg,	R =   90.000 deg
};
P[2460]{
   GP1:
	UF : 0, UT : 6,		CONFIG : 'N U T, 0, 0, 0',
	X =  315.411  mm,	Y =   -101.322  mm,	Z =   -257.120  mm,
	W =  90.000 deg,	P =   0.000 deg,	R =   90.000 deg
};
P[2461]{
   GP1:
	UF : 0, UT : 6,		CONFIG : 'N U T, 0, 0, 0',
	X =  314.845  mm,	Y =   -101.737  mm,	Z =   -257.335  mm,
	W =  90.000 deg,	P =   0.000 deg,	R =   90.000 deg
};
P[2462]{
   GP1:
	UF : 0, UT : 6,		CONFIG : 'N U T, 0, 0, 0',
	X =  312.738  mm,	Y =   -102.880  mm,	Z =   -257.156  mm,
	W =  90.000 deg,	P =   0.000 deg,	R =   90.000 deg
};
P[2463]{
   GP1:
	UF : 0, UT : 6,		CONFIG : 'N U T, 0, 0, 0',
	X =  310.999  mm,	Y =   -103.813  mm,	Z =   -256.983  mm,
	W =  90.000 deg,	P =   0.000 deg,	R =   90.000 deg
};
P[2464]{
   GP1:
	UF : 0, UT : 6,		CONFIG : 'N U T, 0, 0, 0',
	X =  309.607  mm,	Y =   -104.699  mm,	Z =   -257.185  mm,
	W =  90.000 deg,	P =   0.000 deg,	R =   90.000 deg
};
P[2465]{
   GP1:
	UF : 0, UT : 6,		CONFIG : 'N U T, 0, 0, 0',
	X =  306.787  mm,	Y =   -106.316  mm,	Z =   -257.156  mm,
	W =  90.000 deg,	P =   0.000 deg,	R =   90.000 deg
};
P[2466]{
   GP1:
	UF : 0, UT : 6,		CONFIG : 'N U T, 0, 0, 0',
	X =  304.540  mm,	Y =   -107.637  mm,	Z =   -257.214  mm,
	W =  90.000 deg,	P =   0.000 deg,	R =   90.000 deg
};
P[2467]{
   GP1:
	UF : 0, UT : 6,		CONFIG : 'N U T, 0, 0, 0',
	X =  301.156  mm,	Y =   -109.572  mm,	Z =   -257.167  mm,
	W =  90.000 deg,	P =   0.000 deg,	R =   90.000 deg
};
P[2468]{
   GP1:
	UF : 0, UT : 6,		CONFIG : 'N U T, 0, 0, 0',
	X =  297.733  mm,	Y =   -111.447  mm,	Z =   -256.919  mm,
	W =  90.000 deg,	P =   0.000 deg,	R =   90.000 deg
};
P[2469]{
   GP1:
	UF : 0, UT : 6,		CONFIG : 'N U T, 0, 0, 0',
	X =  297.110  mm,	Y =   -111.948  mm,	Z =   -257.266  mm,
	W =  90.000 deg,	P =   0.000 deg,	R =   90.000 deg
};
P[2470]{
   GP1:
	UF : 0, UT : 6,		CONFIG : 'N U T, 0, 0, 0',
	X =  296.219  mm,	Y =   -112.479  mm,	Z =   -257.303  mm,
	W =  90.000 deg,	P =   0.000 deg,	R =   90.000 deg
};
P[2471]{
   GP1:
	UF : 0, UT : 6,		CONFIG : 'N U T, 0, 0, 0',
	X =  295.131  mm,	Y =   -113.009  mm,	Z =   -257.066  mm,
	W =  90.000 deg,	P =   0.000 deg,	R =   90.000 deg
};
P[2472]{
   GP1:
	UF : 0, UT : 6,		CONFIG : 'N U T, 0, 0, 0',
	X =  293.798  mm,	Y =   -113.793  mm,	Z =   -257.100  mm,
	W =  90.000 deg,	P =   0.000 deg,	R =   90.000 deg
};
P[2473]{
   GP1:
	UF : 0, UT : 6,		CONFIG : 'N U T, 0, 0, 0',
	X =  292.780  mm,	Y =   -114.353  mm,	Z =   -257.033  mm,
	W =  90.000 deg,	P =   0.000 deg,	R =   90.000 deg
};
P[2474]{
   GP1:
	UF : 0, UT : 6,		CONFIG : 'N U T, 0, 0, 0',
	X =  291.966  mm,	Y =   -114.917  mm,	Z =   -257.260  mm,
	W =  90.000 deg,	P =   0.000 deg,	R =   90.000 deg
};
P[2475]{
   GP1:
	UF : 0, UT : 6,		CONFIG : 'N U T, 0, 0, 0',
	X =  289.377  mm,	Y =   -116.427  mm,	Z =   -257.298  mm,
	W =  90.000 deg,	P =   0.000 deg,	R =   90.000 deg
};
P[2476]{
   GP1:
	UF : 0, UT : 6,		CONFIG : 'N U T, 0, 0, 0',
	X =  288.003  mm,	Y =   -117.224  mm,	Z =   -257.307  mm,
	W =  90.000 deg,	P =   0.000 deg,	R =   90.000 deg
};
P[2477]{
   GP1:
	UF : 0, UT : 6,		CONFIG : 'N U T, 0, 0, 0',
	X =  286.728  mm,	Y =   -117.988  mm,	Z =   -257.376  mm,
	W =  90.000 deg,	P =   0.000 deg,	R =   90.000 deg
};
P[2478]{
   GP1:
	UF : 0, UT : 6,		CONFIG : 'N U T, 0, 0, 0',
	X =  283.396  mm,	Y =   -119.885  mm,	Z =   -257.309  mm,
	W =  90.000 deg,	P =   0.000 deg,	R =   90.000 deg
};
P[2479]{
   GP1:
	UF : 0, UT : 6,		CONFIG : 'N U T, 0, 0, 0',
	X =  281.063  mm,	Y =   -121.152  mm,	Z =   -257.116  mm,
	W =  90.000 deg,	P =   0.000 deg,	R =   90.000 deg
};
P[2480]{
   GP1:
	UF : 0, UT : 6,		CONFIG : 'N U T, 0, 0, 0',
	X =  277.526  mm,	Y =   -123.234  mm,	Z =   -257.212  mm,
	W =  90.000 deg,	P =   0.000 deg,	R =   90.000 deg
};
P[2481]{
   GP1:
	UF : 0, UT : 6,		CONFIG : 'N U T, 0, 0, 0',
	X =  274.199  mm,	Y =   -125.115  mm,	Z =   -257.115  mm,
	W =  90.000 deg,	P =   0.000 deg,	R =   90.000 deg
};
P[2482]{
   GP1:
	UF : 0, UT : 6,		CONFIG : 'N U T, 0, 0, 0',
	X =  272.661  mm,	Y =   -125.916  mm,	Z =   -256.903  mm,
	W =  90.000 deg,	P =   0.000 deg,	R =   90.000 deg
};
P[2483]{
   GP1:
	UF : 0, UT : 6,		CONFIG : 'N U T, 0, 0, 0',
	X =  271.696  mm,	Y =   -126.637  mm,	Z =   -257.301  mm,
	W =  90.000 deg,	P =   0.000 deg,	R =   90.000 deg
};
P[2484]{
   GP1:
	UF : 0, UT : 6,		CONFIG : 'N U T, 0, 0, 0',
	X =  270.495  mm,	Y =   -127.350  mm,	Z =   -257.349  mm,
	W =  90.000 deg,	P =   0.000 deg,	R =   90.000 deg
};
P[2485]{
   GP1:
	UF : 0, UT : 6,		CONFIG : 'N U T, 0, 0, 0',
	X =  269.035  mm,	Y =   -128.105  mm,	Z =   -257.135  mm,
	W =  90.000 deg,	P =   0.000 deg,	R =   90.000 deg
};
P[2486]{
   GP1:
	UF : 0, UT : 6,		CONFIG : 'N U T, 0, 0, 0',
	X =  268.212  mm,	Y =   -128.636  mm,	Z =   -257.272  mm,
	W =  90.000 deg,	P =   0.000 deg,	R =   90.000 deg
};
P[2487]{
   GP1:
	UF : 0, UT : 6,		CONFIG : 'N U T, 0, 0, 0',
	X =  267.586  mm,	Y =   -128.894  mm,	Z =   -257.020  mm,
	W =  90.000 deg,	P =   0.000 deg,	R =   90.000 deg
};
P[2488]{
   GP1:
	UF : 0, UT : 6,		CONFIG : 'N U T, 0, 0, 0',
	X =  263.716  mm,	Y =   -131.167  mm,	Z =   -257.112  mm,
	W =  90.000 deg,	P =   0.000 deg,	R =   90.000 deg
};
P[2489]{
   GP1:
	UF : 0, UT : 6,		CONFIG : 'N U T, 0, 0, 0',
	X =  261.309  mm,	Y =   -132.493  mm,	Z =   -256.960  mm,
	W =  90.000 deg,	P =   0.000 deg,	R =   90.000 deg
};
P[2490]{
   GP1:
	UF : 0, UT : 6,		CONFIG : 'N U T, 0, 0, 0',
	X =  259.175  mm,	Y =   -133.782  mm,	Z =   -257.096  mm,
	W =  90.000 deg,	P =   0.000 deg,	R =   90.000 deg
};
P[2491]{
   GP1:
	UF : 0, UT : 6,		CONFIG : 'N U T, 0, 0, 0',
	X =  258.310  mm,	Y =   -134.340  mm,	Z =   -257.239  mm,
	W =  90.000 deg,	P =   0.000 deg,	R =   90.000 deg
};
P[2492]{
   GP1:
	UF : 0, UT : 6,		CONFIG : 'N U T, 0, 0, 0',
	X =  257.180  mm,	Y =   -134.989  mm,	Z =   -257.229  mm,
	W =  90.000 deg,	P =   0.000 deg,	R =   90.000 deg
};
P[2493]{
   GP1:
	UF : 0, UT : 6,		CONFIG : 'N U T, 0, 0, 0',
	X =  255.811  mm,	Y =   -135.705  mm,	Z =   -257.049  mm,
	W =  90.000 deg,	P =   0.000 deg,	R =   90.000 deg
};
P[2494]{
   GP1:
	UF : 0, UT : 6,		CONFIG : 'N U T, 0, 0, 0',
	X =  254.069  mm,	Y =   -136.729  mm,	Z =   -257.092  mm,
	W =  90.000 deg,	P =   0.000 deg,	R =   90.000 deg
};
P[2495]{
   GP1:
	UF : 0, UT : 6,		CONFIG : 'N U T, 0, 0, 0',
	X =  251.314  mm,	Y =   -138.374  mm,	Z =   -257.224  mm,
	W =  90.000 deg,	P =   0.000 deg,	R =   90.000 deg
};
P[2496]{
   GP1:
	UF : 0, UT : 6,		CONFIG : 'N U T, 0, 0, 0',
	X =  250.429  mm,	Y =   -138.892  mm,	Z =   -257.242  mm,
	W =  90.000 deg,	P =   0.000 deg,	R =   90.000 deg
};
P[2497]{
   GP1:
	UF : 0, UT : 6,		CONFIG : 'N U T, 0, 0, 0',
	X =  249.298  mm,	Y =   -139.531  mm,	Z =   -257.207  mm,
	W =  90.000 deg,	P =   0.000 deg,	R =   90.000 deg
};
P[2498]{
   GP1:
	UF : 0, UT : 6,		CONFIG : 'N U T, 0, 0, 0',
	X =  247.788  mm,	Y =   -140.299  mm,	Z =   -256.956  mm,
	W =  90.000 deg,	P =   0.000 deg,	R =   90.000 deg
};
P[2499]{
   GP1:
	UF : 0, UT : 6,		CONFIG : 'N U T, 0, 0, 0',
	X =  245.718  mm,	Y =   -141.621  mm,	Z =   -257.262  mm,
	W =  90.000 deg,	P =   0.000 deg,	R =   90.000 deg
};
P[2500]{
   GP1:
	UF : 0, UT : 6,		CONFIG : 'N U T, 0, 0, 0',
	X =  241.441  mm,	Y =   -144.088  mm,	Z =   -257.258  mm,
	W =  90.000 deg,	P =   0.000 deg,	R =   90.000 deg
};
P[2501]{
   GP1:
	UF : 0, UT : 6,		CONFIG : 'N U T, 0, 0, 0',
	X =  240.598  mm,	Y =   -144.556  mm,	Z =   -257.211  mm,
	W =  90.000 deg,	P =   0.000 deg,	R =   90.000 deg
};
P[2502]{
   GP1:
	UF : 0, UT : 6,		CONFIG : 'N U T, 0, 0, 0',
	X =  236.306  mm,	Y =   -147.070  mm,	Z =   -257.298  mm,
	W =  90.000 deg,	P =   0.000 deg,	R =   90.000 deg
};
P[2503]{
   GP1:
	UF : 0, UT : 6,		CONFIG : 'N U T, 0, 0, 0',
	X =  230.880  mm,	Y =   -150.159  mm,	Z =   -257.191  mm,
	W =  90.000 deg,	P =   0.000 deg,	R =   90.000 deg
};
P[2504]{
   GP1:
	UF : 0, UT : 6,		CONFIG : 'N U T, 0, 0, 0',
	X =  229.339  mm,	Y =   -151.055  mm,	Z =   -257.208  mm,
	W =  90.000 deg,	P =   0.000 deg,	R =   90.000 deg
};
P[2505]{
   GP1:
	UF : 0, UT : 6,		CONFIG : 'N U T, 0, 0, 0',
	X =  227.715  mm,	Y =   -151.902  mm,	Z =   -256.988  mm,
	W =  90.000 deg,	P =   0.000 deg,	R =   90.000 deg
};
P[2506]{
   GP1:
	UF : 0, UT : 6,		CONFIG : 'N U T, 0, 0, 0',
	X =  226.793  mm,	Y =   -152.554  mm,	Z =   -257.278  mm,
	W =  90.000 deg,	P =   0.000 deg,	R =   90.000 deg
};
P[2507]{
   GP1:
	UF : 0, UT : 6,		CONFIG : 'N U T, 0, 0, 0',
	X =  226.074  mm,	Y =   -152.941  mm,	Z =   -257.208  mm,
	W =  90.000 deg,	P =   0.000 deg,	R =   90.000 deg
};
P[2508]{
   GP1:
	UF : 0, UT : 6,		CONFIG : 'N U T, 0, 0, 0',
	X =  224.020  mm,	Y =   -154.181  mm,	Z =   -257.340  mm,
	W =  90.000 deg,	P =   0.000 deg,	R =   90.000 deg
};
P[2509]{
   GP1:
	UF : 0, UT : 6,		CONFIG : 'N U T, 0, 0, 0',
	X =  223.395  mm,	Y =   -154.539  mm,	Z =   -257.336  mm,
	W =  90.000 deg,	P =   0.000 deg,	R =   90.000 deg
};
P[2510]{
   GP1:
	UF : 0, UT : 6,		CONFIG : 'N U T, 0, 0, 0',
	X =  220.814  mm,	Y =   -155.913  mm,	Z =   -257.051  mm,
	W =  90.000 deg,	P =   0.000 deg,	R =   90.000 deg
};
P[2511]{
   GP1:
	UF : 0, UT : 6,		CONFIG : 'N U T, 0, 0, 0',
	X =  219.653  mm,	Y =   -156.676  mm,	Z =   -257.277  mm,
	W =  90.000 deg,	P =   0.000 deg,	R =   90.000 deg
};
P[2512]{
   GP1:
	UF : 0, UT : 6,		CONFIG : 'N U T, 0, 0, 0',
	X =  214.862  mm,	Y =   -159.416  mm,	Z =   -257.212  mm,
	W =  90.000 deg,	P =   0.000 deg,	R =   90.000 deg
};
P[2513]{
   GP1:
	UF : 0, UT : 6,		CONFIG : 'N U T, 0, 0, 0',
	X =  211.588  mm,	Y =   -161.279  mm,	Z =   -257.146  mm,
	W =  90.000 deg,	P =   0.000 deg,	R =   90.000 deg
};
P[2514]{
   GP1:
	UF : 0, UT : 6,		CONFIG : 'N U T, 0, 0, 0',
	X =  210.853  mm,	Y =   -161.777  mm,	Z =   -257.324  mm,
	W =  90.000 deg,	P =   0.000 deg,	R =   90.000 deg
};
P[2515]{
   GP1:
	UF : 0, UT : 6,		CONFIG : 'N U T, 0, 0, 0',
	X =  209.201  mm,	Y =   -162.646  mm,	Z =   -257.119  mm,
	W =  90.000 deg,	P =   0.000 deg,	R =   90.000 deg
};
P[2516]{
   GP1:
	UF : 0, UT : 6,		CONFIG : 'N U T, 0, 0, 0',
	X =  208.313  mm,	Y =   -163.229  mm,	Z =   -257.288  mm,
	W =  90.000 deg,	P =   0.000 deg,	R =   90.000 deg
};
P[2517]{
   GP1:
	UF : 0, UT : 6,		CONFIG : 'N U T, 0, 0, 0',
	X =  207.070  mm,	Y =   -163.985  mm,	Z =   -257.382  mm,
	W =  90.000 deg,	P =   0.000 deg,	R =   90.000 deg
};
P[2518]{
   GP1:
	UF : 0, UT : 6,		CONFIG : 'N U T, 0, 0, 0',
	X =  204.070  mm,	Y =   -165.530  mm,	Z =   -256.928  mm,
	W =  90.000 deg,	P =   0.000 deg,	R =   90.000 deg
};
P[2519]{
   GP1:
	UF : 0, UT : 6,		CONFIG : 'N U T, 0, 0, 0',
	X =  202.708  mm,	Y =   -166.304  mm,	Z =   -256.897  mm,
	W =  90.000 deg,	P =   0.000 deg,	R =   90.000 deg
};
P[2520]{
   GP1:
	UF : 0, UT : 6,		CONFIG : 'N U T, 0, 0, 0',
	X =  200.710  mm,	Y =   -167.561  mm,	Z =   -257.148  mm,
	W =  90.000 deg,	P =   0.000 deg,	R =   90.000 deg
};
P[2521]{
   GP1:
	UF : 0, UT : 6,		CONFIG : 'N U T, 0, 0, 0',
	X =  199.405  mm,	Y =   -168.208  mm,	Z =   -256.889  mm,
	W =  90.000 deg,	P =   0.000 deg,	R =   90.000 deg
};
P[2522]{
   GP1:
	UF : 0, UT : 6,		CONFIG : 'N U T, 0, 0, 0',
	X =  198.612  mm,	Y =   -168.864  mm,	Z =   -257.370  mm,
	W =  90.000 deg,	P =   0.000 deg,	R =   90.000 deg
};
P[2523]{
   GP1:
	UF : 0, UT : 6,		CONFIG : 'N U T, 0, 0, 0',
	X =  195.171  mm,	Y =   -170.683  mm,	Z =   -256.965  mm,
	W =  90.000 deg,	P =   0.000 deg,	R =   90.000 deg
};
P[2524]{
   GP1:
	UF : 0, UT : 6,		CONFIG : 'N U T, 0, 0, 0',
	X =  194.418  mm,	Y =   -171.181  mm,	Z =   -257.116  mm,
	W =  90.000 deg,	P =   0.000 deg,	R =   90.000 deg
};
P[2525]{
   GP1:
	UF : 0, UT : 6,		CONFIG : 'N U T, 0, 0, 0',
	X =  192.248  mm,	Y =   -172.428  mm,	Z =   -257.105  mm,
	W =  90.000 deg,	P =   0.000 deg,	R =   90.000 deg
};
P[2526]{
   GP1:
	UF : 0, UT : 6,		CONFIG : 'N U T, 0, 0, 0',
	X =  190.442  mm,	Y =   -173.511  mm,	Z =   -257.200  mm,
	W =  90.000 deg,	P =   0.000 deg,	R =   90.000 deg
};
P[2527]{
   GP1:
	UF : 0, UT : 6,		CONFIG : 'N U T, 0, 0, 0',
	X =  189.315  mm,	Y =   -174.097  mm,	Z =   -257.044  mm,
	W =  90.000 deg,	P =   0.000 deg,	R =   90.000 deg
};
P[2528]{
   GP1:
	UF : 0, UT : 6,		CONFIG : 'N U T, 0, 0, 0',
	X =  186.556  mm,	Y =   -175.716  mm,	Z =   -257.109  mm,
	W =  90.000 deg,	P =   0.000 deg,	R =   90.000 deg
};
P[2529]{
   GP1:
	UF : 0, UT : 6,		CONFIG : 'N U T, 0, 0, 0',
	X =  185.928  mm,	Y =   -176.024  mm,	Z =   -256.975  mm,
	W =  90.000 deg,	P =   0.000 deg,	R =   90.000 deg
};
P[2530]{
   GP1:
	UF : 0, UT : 6,		CONFIG : 'N U T, 0, 0, 0',
	X =  183.536  mm,	Y =   -177.407  mm,	Z =   -256.978  mm,
	W =  90.000 deg,	P =   0.000 deg,	R =   90.000 deg
};
P[2531]{
   GP1:
	UF : 0, UT : 6,		CONFIG : 'N U T, 0, 0, 0',
	X =  181.508  mm,	Y =   -178.677  mm,	Z =   -257.218  mm,
	W =  90.000 deg,	P =   0.000 deg,	R =   90.000 deg
};
P[2532]{
   GP1:
	UF : 0, UT : 6,		CONFIG : 'N U T, 0, 0, 0',
	X =  180.157  mm,	Y =   -179.515  mm,	Z =   -257.360  mm,
	W =  90.000 deg,	P =   0.000 deg,	R =   90.000 deg
};
P[2533]{
   GP1:
	UF : 0, UT : 6,		CONFIG : 'N U T, 0, 0, 0',
	X =  178.903  mm,	Y =   -180.053  mm,	Z =   -256.909  mm,
	W =  90.000 deg,	P =   0.000 deg,	R =   90.000 deg
};
P[2534]{
   GP1:
	UF : 0, UT : 6,		CONFIG : 'N U T, 0, 0, 0',
	X =  178.429  mm,	Y =   -180.483  mm,	Z =   -257.290  mm,
	W =  90.000 deg,	P =   0.000 deg,	R =   90.000 deg
};
P[2535]{
   GP1:
	UF : 0, UT : 6,		CONFIG : 'N U T, 0, 0, 0',
	X =  177.666  mm,	Y =   -180.855  mm,	Z =   -257.119  mm,
	W =  90.000 deg,	P =   0.000 deg,	R =   90.000 deg
};
P[2536]{
   GP1:
	UF : 0, UT : 6,		CONFIG : 'N U T, 0, 0, 0',
	X =  176.659  mm,	Y =   -181.494  mm,	Z =   -257.262  mm,
	W =  90.000 deg,	P =   0.000 deg,	R =   90.000 deg
};
P[2537]{
   GP1:
	UF : 0, UT : 6,		CONFIG : 'N U T, 0, 0, 0',
	X =  172.885  mm,	Y =   -183.687  mm,	Z =   -257.294  mm,
	W =  90.000 deg,	P =   0.000 deg,	R =   90.000 deg
};
P[2538]{
   GP1:
	UF : 0, UT : 6,		CONFIG : 'N U T, 0, 0, 0',
	X =  170.695  mm,	Y =   -184.819  mm,	Z =   -256.974  mm,
	W =  90.000 deg,	P =   0.000 deg,	R =   90.000 deg
};
P[2539]{
   GP1:
	UF : 0, UT : 6,		CONFIG : 'N U T, 0, 0, 0',
	X =  168.152  mm,	Y =   -186.375  mm,	Z =   -257.186  mm,
	W =  90.000 deg,	P =   0.000 deg,	R =   90.000 deg
};
P[2540]{
   GP1:
	UF : 0, UT : 6,		CONFIG : 'N U T, 0, 0, 0',
	X =  165.761  mm,	Y =   -187.745  mm,	Z =   -257.160  mm,
	W =  90.000 deg,	P =   0.000 deg,	R =   90.000 deg
};
P[2541]{
   GP1:
	UF : 0, UT : 6,		CONFIG : 'N U T, 0, 0, 0',
	X =  164.162  mm,	Y =   -188.630  mm,	Z =   -257.070  mm,
	W =  90.000 deg,	P =   0.000 deg,	R =   90.000 deg
};
P[2542]{
   GP1:
	UF : 0, UT : 6,		CONFIG : 'N U T, 0, 0, 0',
	X =  162.369  mm,	Y =   -189.720  mm,	Z =   -257.200  mm,
	W =  90.000 deg,	P =   0.000 deg,	R =   90.000 deg
};
P[2543]{
   GP1:
	UF : 0, UT : 6,		CONFIG : 'N U T, 0, 0, 0',
	X =  158.313  mm,	Y =   -192.117  mm,	Z =   -257.334  mm,
	W =  90.000 deg,	P =   0.000 deg,	R =   90.000 deg
};
P[2544]{
   GP1:
	UF : 0, UT : 6,		CONFIG : 'N U T, 0, 0, 0',
	X =  156.553  mm,	Y =   -193.138  mm,	Z =   -257.344  mm,
	W =  90.000 deg,	P =   0.000 deg,	R =   90.000 deg
};
P[2545]{
   GP1:
	UF : 0, UT : 6,		CONFIG : 'N U T, 0, 0, 0',
	X =  154.553  mm,	Y =   -194.211  mm,	Z =   -257.147  mm,
	W =  90.000 deg,	P =   0.000 deg,	R =   90.000 deg
};
P[2546]{
   GP1:
	UF : 0, UT : 6,		CONFIG : 'N U T, 0, 0, 0',
	X =  153.108  mm,	Y =   -195.114  mm,	Z =   -257.313  mm,
	W =  90.000 deg,	P =   0.000 deg,	R =   90.000 deg
};
P[2547]{
   GP1:
	UF : 0, UT : 6,		CONFIG : 'N U T, 0, 0, 0',
	X =  151.694  mm,	Y =   -195.895  mm,	Z =   -257.227  mm,
	W =  90.000 deg,	P =   0.000 deg,	R =   90.000 deg
};
P[2548]{
   GP1:
	UF : 0, UT : 6,		CONFIG : 'N U T, 0, 0, 0',
	X =  149.080  mm,	Y =   -197.376  mm,	Z =   -257.160  mm,
	W =  90.000 deg,	P =   0.000 deg,	R =   90.000 deg
};
P[2549]{
   GP1:
	UF : 0, UT : 6,		CONFIG : 'N U T, 0, 0, 0',
	X =  147.973  mm,	Y =   -198.063  mm,	Z =   -257.277  mm,
	W =  90.000 deg,	P =   0.000 deg,	R =   90.000 deg
};
P[2550]{
   GP1:
	UF : 0, UT : 6,		CONFIG : 'N U T, 0, 0, 0',
	X =  147.033  mm,	Y =   -198.503  mm,	Z =   -257.026  mm,
	W =  90.000 deg,	P =   0.000 deg,	R =   90.000 deg
};
P[2551]{
   GP1:
	UF : 0, UT : 6,		CONFIG : 'N U T, 0, 0, 0',
	X =  143.928  mm,	Y =   -200.377  mm,	Z =   -257.225  mm,
	W =  90.000 deg,	P =   0.000 deg,	R =   90.000 deg
};
P[2552]{
   GP1:
	UF : 0, UT : 6,		CONFIG : 'N U T, 0, 0, 0',
	X =  143.166  mm,	Y =   -200.877  mm,	Z =   -257.371  mm,
	W =  90.000 deg,	P =   0.000 deg,	R =   90.000 deg
};
P[2553]{
   GP1:
	UF : 0, UT : 6,		CONFIG : 'N U T, 0, 0, 0',
	X =  137.744  mm,	Y =   -203.978  mm,	Z =   -257.296  mm,
	W =  90.000 deg,	P =   0.000 deg,	R =   90.000 deg
};
P[2554]{
   GP1:
	UF : 0, UT : 6,		CONFIG : 'N U T, 0, 0, 0',
	X =  136.696  mm,	Y =   -204.550  mm,	Z =   -257.217  mm,
	W =  90.000 deg,	P =   0.000 deg,	R =   90.000 deg
};
P[2555]{
   GP1:
	UF : 0, UT : 6,		CONFIG : 'N U T, 0, 0, 0',
	X =  131.945  mm,	Y =   -207.203  mm,	Z =   -256.997  mm,
	W =  90.000 deg,	P =   0.000 deg,	R =   90.000 deg
};
P[2556]{
   GP1:
	UF : 0, UT : 6,		CONFIG : 'N U T, 0, 0, 0',
	X =  129.524  mm,	Y =   -208.631  mm,	Z =   -257.072  mm,
	W =  90.000 deg,	P =   0.000 deg,	R =   90.000 deg
};
P[2557]{
   GP1:
	UF : 0, UT : 6,		CONFIG : 'N U T, 0, 0, 0',
	X =  127.779  mm,	Y =   -209.624  mm,	Z =   -257.037  mm,
	W =  90.000 deg,	P =   0.000 deg,	R =   90.000 deg
};
P[2558]{
   GP1:
	UF : 0, UT : 6,		CONFIG : 'N U T, 0, 0, 0',
	X =  126.158  mm,	Y =   -210.556  mm,	Z =   -257.026  mm,
	W =  90.000 deg,	P =   0.000 deg,	R =   90.000 deg
};
P[2559]{
   GP1:
	UF : 0, UT : 6,		CONFIG : 'N U T, 0, 0, 0',
	X =  122.642  mm,	Y =   -212.657  mm,	Z =   -257.199  mm,
	W =  90.000 deg,	P =   0.000 deg,	R =   90.000 deg
};
P[2560]{
   GP1:
	UF : 0, UT : 6,		CONFIG : 'N U T, 0, 0, 0',
	X =  121.983  mm,	Y =   -213.080  mm,	Z =   -257.302  mm,
	W =  90.000 deg,	P =   0.000 deg,	R =   90.000 deg
};
P[2561]{
   GP1:
	UF : 0, UT : 6,		CONFIG : 'N U T, 0, 0, 0',
	X =  121.007  mm,	Y =   -213.533  mm,	Z =   -257.033  mm,
	W =  90.000 deg,	P =   0.000 deg,	R =   90.000 deg
};
P[2562]{
   GP1:
	UF : 0, UT : 6,		CONFIG : 'N U T, 0, 0, 0',
	X =  118.998  mm,	Y =   -214.697  mm,	Z =   -257.044  mm,
	W =  90.000 deg,	P =   0.000 deg,	R =   90.000 deg
};
P[2563]{
   GP1:
	UF : 0, UT : 6,		CONFIG : 'N U T, 0, 0, 0',
	X =  116.054  mm,	Y =   -214.009  mm,	Z =   -251.246  mm,
	W =  90.000 deg,	P =   0.000 deg,	R =   90.000 deg
};
P[2564]{
   GP1:
	UF : 0, UT : 6,		CONFIG : 'N U T, 0, 0, 0',
	X =  115.305  mm,	Y =   -214.349  mm,	Z =   -251.023  mm,
	W =  90.000 deg,	P =   0.000 deg,	R =   90.000 deg
};
P[2565]{
   GP1:
	UF : 0, UT : 6,		CONFIG : 'N U T, 0, 0, 0',
	X =  114.750  mm,	Y =   -214.842  mm,	Z =   -251.441  mm,
	W =  90.000 deg,	P =   0.000 deg,	R =   90.000 deg
};
P[2566]{
   GP1:
	UF : 0, UT : 6,		CONFIG : 'N U T, 0, 0, 0',
	X =  112.482  mm,	Y =   -216.000  mm,	Z =   -251.075  mm,
	W =  90.000 deg,	P =   0.000 deg,	R =   90.000 deg
};
P[2567]{
   GP1:
	UF : 0, UT : 6,		CONFIG : 'N U T, 0, 0, 0',
	X =  110.818  mm,	Y =   -217.112  mm,	Z =   -251.441  mm,
	W =  90.000 deg,	P =   0.000 deg,	R =   90.000 deg
};
P[2568]{
   GP1:
	UF : 0, UT : 6,		CONFIG : 'N U T, 0, 0, 0',
	X =  108.986  mm,	Y =   -218.173  mm,	Z =   -251.449  mm,
	W =  90.000 deg,	P =   0.000 deg,	R =   90.000 deg
};
P[2569]{
   GP1:
	UF : 0, UT : 6,		CONFIG : 'N U T, 0, 0, 0',
	X =  106.975  mm,	Y =   -219.287  mm,	Z =   -251.335  mm,
	W =  90.000 deg,	P =   0.000 deg,	R =   90.000 deg
};
P[2570]{
   GP1:
	UF : 0, UT : 6,		CONFIG : 'N U T, 0, 0, 0',
	X =  102.759  mm,	Y =   -221.774  mm,	Z =   -251.464  mm,
	W =  90.000 deg,	P =   0.000 deg,	R =   90.000 deg
};
P[2571]{
   GP1:
	UF : 0, UT : 6,		CONFIG : 'N U T, 0, 0, 0',
	X =  101.224  mm,	Y =   -222.643  mm,	Z =   -251.421  mm,
	W =  90.000 deg,	P =   0.000 deg,	R =   90.000 deg
};
P[2572]{
   GP1:
	UF : 0, UT : 6,		CONFIG : 'N U T, 0, 0, 0',
	X =  99.448  mm,	Y =   -223.549  mm,	Z =   -251.130  mm,
	W =  90.000 deg,	P =   0.000 deg,	R =   90.000 deg
};
P[2573]{
   GP1:
	UF : 0, UT : 6,		CONFIG : 'N U T, 0, 0, 0',
	X =  97.555  mm,	Y =   -224.706  mm,	Z =   -251.287  mm,
	W =  90.000 deg,	P =   0.000 deg,	R =   90.000 deg
};
P[2574]{
   GP1:
	UF : 0, UT : 6,		CONFIG : 'N U T, 0, 0, 0',
	X =  97.015  mm,	Y =   -225.111  mm,	Z =   -251.512  mm,
	W =  90.000 deg,	P =   0.000 deg,	R =   90.000 deg
};
P[2575]{
   GP1:
	UF : 0, UT : 6,		CONFIG : 'N U T, 0, 0, 0',
	X =  93.650  mm,	Y =   -227.025  mm,	Z =   -251.442  mm,
	W =  90.000 deg,	P =   0.000 deg,	R =   90.000 deg
};
P[2576]{
   GP1:
	UF : 0, UT : 6,		CONFIG : 'N U T, 0, 0, 0',
	X =  91.936  mm,	Y =   -228.021  mm,	Z =   -251.457  mm,
	W =  90.000 deg,	P =   0.000 deg,	R =   90.000 deg
};
P[2577]{
   GP1:
	UF : 0, UT : 6,		CONFIG : 'N U T, 0, 0, 0',
	X =  91.024  mm,	Y =   -228.501  mm,	Z =   -251.346  mm,
	W =  90.000 deg,	P =   0.000 deg,	R =   90.000 deg
};
P[2578]{
   GP1:
	UF : 0, UT : 6,		CONFIG : 'N U T, 0, 0, 0',
	X =  89.278  mm,	Y =   -229.472  mm,	Z =   -251.256  mm,
	W =  90.000 deg,	P =   0.000 deg,	R =   90.000 deg
};
P[2579]{
   GP1:
	UF : 0, UT : 6,		CONFIG : 'N U T, 0, 0, 0',
	X =  86.740  mm,	Y =   -230.846  mm,	Z =   -251.034  mm,
	W =  90.000 deg,	P =   0.000 deg,	R =   90.000 deg
};
P[2580]{
   GP1:
	UF : 0, UT : 6,		CONFIG : 'N U T, 0, 0, 0',
	X =  83.701  mm,	Y =   -232.723  mm,	Z =   -251.330  mm,
	W =  90.000 deg,	P =   0.000 deg,	R =   90.000 deg
};
P[2581]{
   GP1:
	UF : 0, UT : 6,		CONFIG : 'N U T, 0, 0, 0',
	X =  81.905  mm,	Y =   -233.763  mm,	Z =   -251.338  mm,
	W =  90.000 deg,	P =   0.000 deg,	R =   90.000 deg
};
P[2582]{
   GP1:
	UF : 0, UT : 6,		CONFIG : 'N U T, 0, 0, 0',
	X =  80.406  mm,	Y =   -234.585  mm,	Z =   -251.228  mm,
	W =  90.000 deg,	P =   0.000 deg,	R =   90.000 deg
};
P[2583]{
   GP1:
	UF : 0, UT : 6,		CONFIG : 'N U T, 0, 0, 0',
	X =  79.799  mm,	Y =   -234.985  mm,	Z =   -251.351  mm,
	W =  90.000 deg,	P =   0.000 deg,	R =   90.000 deg
};
P[2584]{
   GP1:
	UF : 0, UT : 6,		CONFIG : 'N U T, 0, 0, 0',
	X =  79.236  mm,	Y =   -235.338  mm,	Z =   -251.419  mm,
	W =  90.000 deg,	P =   0.000 deg,	R =   90.000 deg
};
P[2585]{
   GP1:
	UF : 0, UT : 6,		CONFIG : 'N U T, 0, 0, 0',
	X =  74.732  mm,	Y =   -237.968  mm,	Z =   -251.489  mm,
	W =  90.000 deg,	P =   0.000 deg,	R =   90.000 deg
};
P[2586]{
   GP1:
	UF : 0, UT : 6,		CONFIG : 'N U T, 0, 0, 0',
	X =  72.064  mm,	Y =   -239.480  mm,	Z =   -251.422  mm,
	W =  90.000 deg,	P =   0.000 deg,	R =   90.000 deg
};
P[2587]{
   GP1:
	UF : 0, UT : 6,		CONFIG : 'N U T, 0, 0, 0',
	X =  71.290  mm,	Y =   -239.858  mm,	Z =   -251.254  mm,
	W =  90.000 deg,	P =   0.000 deg,	R =   90.000 deg
};
P[2588]{
   GP1:
	UF : 0, UT : 6,		CONFIG : 'N U T, 0, 0, 0',
	X =  70.531  mm,	Y =   -240.355  mm,	Z =   -251.397  mm,
	W =  90.000 deg,	P =   0.000 deg,	R =   90.000 deg
};
P[2589]{
   GP1:
	UF : 0, UT : 6,		CONFIG : 'N U T, 0, 0, 0',
	X =  69.219  mm,	Y =   -241.070  mm,	Z =   -251.292  mm,
	W =  90.000 deg,	P =   0.000 deg,	R =   90.000 deg
};
P[2590]{
   GP1:
	UF : 0, UT : 6,		CONFIG : 'N U T, 0, 0, 0',
	X =  66.598  mm,	Y =   -242.625  mm,	Z =   -251.393  mm,
	W =  90.000 deg,	P =   0.000 deg,	R =   90.000 deg
};
P[2591]{
   GP1:
	UF : 0, UT : 6,		CONFIG : 'N U T, 0, 0, 0',
	X =  61.580  mm,	Y =   -245.540  mm,	Z =   -251.438  mm,
	W =  90.000 deg,	P =   0.000 deg,	R =   90.000 deg
};
P[2592]{
   GP1:
	UF : 0, UT : 6,		CONFIG : 'N U T, 0, 0, 0',
	X =  56.948  mm,	Y =   -248.218  mm,	Z =   -251.444  mm,
	W =  90.000 deg,	P =   0.000 deg,	R =   90.000 deg
};
P[2593]{
   GP1:
	UF : 0, UT : 6,		CONFIG : 'N U T, 0, 0, 0',
	X =  55.361  mm,	Y =   -249.103  mm,	Z =   -251.370  mm,
	W =  90.000 deg,	P =   0.000 deg,	R =   90.000 deg
};
P[2594]{
   GP1:
	UF : 0, UT : 6,		CONFIG : 'N U T, 0, 0, 0',
	X =  49.449  mm,	Y =   -252.432  mm,	Z =   -251.164  mm,
	W =  90.000 deg,	P =   0.000 deg,	R =   90.000 deg
};
P[2595]{
   GP1:
	UF : 0, UT : 6,		CONFIG : 'N U T, 0, 0, 0',
	X =  48.557  mm,	Y =   -253.008  mm,	Z =   -251.314  mm,
	W =  90.000 deg,	P =   0.000 deg,	R =   90.000 deg
};
P[2596]{
   GP1:
	UF : 0, UT : 6,		CONFIG : 'N U T, 0, 0, 0',
	X =  45.342  mm,	Y =   -254.837  mm,	Z =   -251.246  mm,
	W =  90.000 deg,	P =   0.000 deg,	R =   90.000 deg
};
P[2597]{
   GP1:
	UF : 0, UT : 6,		CONFIG : 'N U T, 0, 0, 0',
	X =  41.417  mm,	Y =   -257.192  mm,	Z =   -251.460  mm,
	W =  90.000 deg,	P =   0.000 deg,	R =   90.000 deg
};
P[2598]{
   GP1:
	UF : 0, UT : 6,		CONFIG : 'N U T, 0, 0, 0',
	X =  39.281  mm,	Y =   -258.352  mm,	Z =   -251.284  mm,
	W =  90.000 deg,	P =   0.000 deg,	R =   90.000 deg
};
P[2599]{
   GP1:
	UF : 0, UT : 6,		CONFIG : 'N U T, 0, 0, 0',
	X =  36.351  mm,	Y =   -259.936  mm,	Z =   -251.022  mm,
	W =  90.000 deg,	P =   0.000 deg,	R =   90.000 deg
};
P[2600]{
   GP1:
	UF : 0, UT : 6,		CONFIG : 'N U T, 0, 0, 0',
	X =  35.617  mm,	Y =   -260.537  mm,	Z =   -251.451  mm,
	W =  90.000 deg,	P =   0.000 deg,	R =   90.000 deg
};
P[2601]{
   GP1:
	UF : 0, UT : 6,		CONFIG : 'N U T, 0, 0, 0',
	X =  34.883  mm,	Y =   -260.943  mm,	Z =   -251.408  mm,
	W =  90.000 deg,	P =   0.000 deg,	R =   90.000 deg
};
P[2602]{
   GP1:
	UF : 0, UT : 6,		CONFIG : 'N U T, 0, 0, 0',
	X =  33.349  mm,	Y =   -261.738  mm,	Z =   -251.190  mm,
	W =  90.000 deg,	P =   0.000 deg,	R =   90.000 deg
};
P[2603]{
   GP1:
	UF : 0, UT : 6,		CONFIG : 'N U T, 0, 0, 0',
	X =  30.827  mm,	Y =   -263.247  mm,	Z =   -251.317  mm,
	W =  90.000 deg,	P =   0.000 deg,	R =   90.000 deg
};
P[2604]{
   GP1:
	UF : 0, UT : 6,		CONFIG : 'N U T, 0, 0, 0',
	X =  29.944  mm,	Y =   -263.698  mm,	Z =   -251.175  mm,
	W =  90.000 deg,	P =   0.000 deg,	R =   90.000 deg
};
P[2605]{
   GP1:
	UF : 0, UT : 6,		CONFIG : 'N U T, 0, 0, 0',
	X =  29.314  mm,	Y =   -264.095  mm,	Z =   -251.256  mm,
	W =  90.000 deg,	P =   0.000 deg,	R =   90.000 deg
};
P[2606]{
   GP1:
	UF : 0, UT : 6,		CONFIG : 'N U T, 0, 0, 0',
	X =  26.620  mm,	Y =   -265.687  mm,	Z =   -251.343  mm,
	W =  90.000 deg,	P =   0.000 deg,	R =   90.000 deg
};
P[2607]{
   GP1:
	UF : 0, UT : 6,		CONFIG : 'N U T, 0, 0, 0',
	X =  25.820  mm,	Y =   -266.096  mm,	Z =   -251.217  mm,
	W =  90.000 deg,	P =   0.000 deg,	R =   90.000 deg
};
P[2608]{
   GP1:
	UF : 0, UT : 6,		CONFIG : 'N U T, 0, 0, 0',
	X =  25.222  mm,	Y =   -266.527  mm,	Z =   -251.421  mm,
	W =  90.000 deg,	P =   0.000 deg,	R =   90.000 deg
};
P[2609]{
   GP1:
	UF : 0, UT : 6,		CONFIG : 'N U T, 0, 0, 0',
	X =  21.283  mm,	Y =   -268.638  mm,	Z =   -251.026  mm,
	W =  90.000 deg,	P =   0.000 deg,	R =   90.000 deg
};
P[2610]{
   GP1:
	UF : 0, UT : 6,		CONFIG : 'N U T, 0, 0, 0',
	X =  17.862  mm,	Y =   -270.738  mm,	Z =   -251.328  mm,
	W =  90.000 deg,	P =   0.000 deg,	R =   90.000 deg
};
P[2611]{
   GP1:
	UF : 0, UT : 6,		CONFIG : 'N U T, 0, 0, 0',
	X =  17.242  mm,	Y =   -270.987  mm,	Z =   -251.065  mm,
	W =  90.000 deg,	P =   0.000 deg,	R =   90.000 deg
};
P[2612]{
   GP1:
	UF : 0, UT : 6,		CONFIG : 'N U T, 0, 0, 0',
	X =  16.617  mm,	Y =   -271.468  mm,	Z =   -251.357  mm,
	W =  90.000 deg,	P =   0.000 deg,	R =   90.000 deg
};
P[2613]{
   GP1:
	UF : 0, UT : 6,		CONFIG : 'N U T, 0, 0, 0',
	X =  15.599  mm,	Y =   -271.997  mm,	Z =   -251.212  mm,
	W =  90.000 deg,	P =   0.000 deg,	R =   90.000 deg
};
P[2614]{
   GP1:
	UF : 0, UT : 6,		CONFIG : 'N U T, 0, 0, 0',
	X =  14.152  mm,	Y =   -272.893  mm,	Z =   -251.362  mm,
	W =  90.000 deg,	P =   0.000 deg,	R =   90.000 deg
};
P[2615]{
   GP1:
	UF : 0, UT : 6,		CONFIG : 'N U T, 0, 0, 0',
	X =  12.772  mm,	Y =   -273.693  mm,	Z =   -251.369  mm,
	W =  90.000 deg,	P =   0.000 deg,	R =   90.000 deg
};
P[2616]{
   GP1:
	UF : 0, UT : 6,		CONFIG : 'N U T, 0, 0, 0',
	X =  8.513  mm,	Y =   -276.151  mm,	Z =   -251.368  mm,
	W =  90.000 deg,	P =   0.000 deg,	R =   90.000 deg
};
P[2617]{
   GP1:
	UF : 0, UT : 6,		CONFIG : 'N U T, 0, 0, 0',
	X =  6.111  mm,	Y =   -277.485  mm,	Z =   -251.236  mm,
	W =  90.000 deg,	P =   0.000 deg,	R =   90.000 deg
};
P[2618]{
   GP1:
	UF : 0, UT : 6,		CONFIG : 'N U T, 0, 0, 0',
	X =  4.557  mm,	Y =   -278.430  mm,	Z =   -251.353  mm,
	W =  90.000 deg,	P =   0.000 deg,	R =   90.000 deg
};
P[2619]{
   GP1:
	UF : 0, UT : 6,		CONFIG : 'N U T, 0, 0, 0',
	X =  2.420  mm,	Y =   -279.679  mm,	Z =   -251.389  mm,
	W =  90.000 deg,	P =   0.000 deg,	R =   90.000 deg
};
P[2620]{
   GP1:
	UF : 0, UT : 6,		CONFIG : 'N U T, 0, 0, 0',
	X =  -0.569  mm,	Y =   -281.268  mm,	Z =   -251.058  mm,
	W =  90.000 deg,	P =   0.000 deg,	R =   90.000 deg
};
P[2621]{
   GP1:
	UF : 0, UT : 6,		CONFIG : 'N U T, 0, 0, 0',
	X =  -1.720  mm,	Y =   -282.009  mm,	Z =   -251.243  mm,
	W =  90.000 deg,	P =   0.000 deg,	R =   90.000 deg
};
P[2622]{
   GP1:
	UF : 0, UT : 6,		CONFIG : 'N U T, 0, 0, 0',
	X =  -5.066  mm,	Y =   -284.045  mm,	Z =   -251.496  mm,
	W =  90.000 deg,	P =   0.000 deg,	R =   90.000 deg
};
P[2623]{
   GP1:
	UF : 0, UT : 6,		CONFIG : 'N U T, 0, 0, 0',
	X =  -8.934  mm,	Y =   -286.209  mm,	Z =   -251.328  mm,
	W =  90.000 deg,	P =   0.000 deg,	R =   90.000 deg
};
P[2624]{
   GP1:
	UF : 0, UT : 6,		CONFIG : 'N U T, 0, 0, 0',
	X =  -9.772  mm,	Y =   -286.686  mm,	Z =   -251.314  mm,
	W =  90.000 deg,	P =   0.000 deg,	R =   90.000 deg
};
P[2625]{
   GP1:
	UF : 0, UT : 6,		CONFIG : 'N U T, 0, 0, 0',
	X =  -11.637  mm,	Y =   -287.720  mm,	Z =   -251.209  mm,
	W =  90.000 deg,	P =   0.000 deg,	R =   90.000 deg
};
P[2626]{
   GP1:
	UF : 0, UT : 6,		CONFIG : 'N U T, 0, 0, 0',
	X =  -12.239  mm,	Y =   -287.989  mm,	Z =   -251.017  mm,
	W =  90.000 deg,	P =   0.000 deg,	R =   90.000 deg
};
P[2627]{
   GP1:
	UF : 0, UT : 6,		CONFIG : 'N U T, 0, 0, 0',
	X =  -13.240  mm,	Y =   -288.748  mm,	Z =   -251.453  mm,
	W =  90.000 deg,	P =   0.000 deg,	R =   90.000 deg
};
P[2628]{
   GP1:
	UF : 0, UT : 6,		CONFIG : 'N U T, 0, 0, 0',
	X =  -14.593  mm,	Y =   -289.477  mm,	Z =   -251.329  mm,
	W =  90.000 deg,	P =   0.000 deg,	R =   90.000 deg
};
P[2629]{
   GP1:
	UF : 0, UT : 6,		CONFIG : 'N U T, 0, 0, 0',
	X =  -18.470  mm,	Y =   -291.678  mm,	Z =   -251.237  mm,
	W =  90.000 deg,	P =   0.000 deg,	R =   90.000 deg
};
P[2630]{
   GP1:
	UF : 0, UT : 6,		CONFIG : 'N U T, 0, 0, 0',
	X =  -19.590  mm,	Y =   -292.298  mm,	Z =   -251.173  mm,
	W =  90.000 deg,	P =   0.000 deg,	R =   90.000 deg
};
P[2631]{
   GP1:
	UF : 0, UT : 6,		CONFIG : 'N U T, 0, 0, 0',
	X =  -21.641  mm,	Y =   -293.543  mm,	Z =   -251.320  mm,
	W =  90.000 deg,	P =   0.000 deg,	R =   90.000 deg
};
P[2632]{
   GP1:
	UF : 0, UT : 6,		CONFIG : 'N U T, 0, 0, 0',
	X =  -22.449  mm,	Y =   -293.970  mm,	Z =   -251.223  mm,
	W =  90.000 deg,	P =   0.000 deg,	R =   90.000 deg
};
P[2633]{
   GP1:
	UF : 0, UT : 6,		CONFIG : 'N U T, 0, 0, 0',
	X =  -24.294  mm,	Y =   -295.043  mm,	Z =   -251.244  mm,
	W =  90.000 deg,	P =   0.000 deg,	R =   90.000 deg
};
P[2634]{
   GP1:
	UF : 0, UT : 6,		CONFIG : 'N U T, 0, 0, 0',
	X =  -29.305  mm,	Y =   -297.952  mm,	Z =   -251.281  mm,
	W =  90.000 deg,	P =   0.000 deg,	R =   90.000 deg
};
P[2635]{
   GP1:
	UF : 0, UT : 6,		CONFIG : 'N U T, 0, 0, 0',
	X =  -30.830  mm,	Y =   -298.905  mm,	Z =   -251.457  mm,
	W =  90.000 deg,	P =   0.000 deg,	R =   90.000 deg
};
P[2636]{
   GP1:
	UF : 0, UT : 6,		CONFIG : 'N U T, 0, 0, 0',
	X =  -31.945  mm,	Y =   -299.523  mm,	Z =   -251.395  mm,
	W =  90.000 deg,	P =   0.000 deg,	R =   90.000 deg
};
P[2637]{
   GP1:
	UF : 0, UT : 6,		CONFIG : 'N U T, 0, 0, 0',
	X =  -33.377  mm,	Y =   -300.352  mm,	Z =   -251.401  mm,
	W =  90.000 deg,	P =   0.000 deg,	R =   90.000 deg
};
P[2638]{
   GP1:
	UF : 0, UT : 6,		CONFIG : 'N U T, 0, 0, 0',
	X =  -35.442  mm,	Y =   -301.530  mm,	Z =   -251.365  mm,
	W =  90.000 deg,	P =   0.000 deg,	R =   90.000 deg
};
P[2639]{
   GP1:
	UF : 0, UT : 6,		CONFIG : 'N U T, 0, 0, 0',
	X =  -36.250  mm,	Y =   -301.892  mm,	Z =   -251.112  mm,
	W =  90.000 deg,	P =   0.000 deg,	R =   90.000 deg
};
P[2640]{
   GP1:
	UF : 0, UT : 6,		CONFIG : 'N U T, 0, 0, 0',
	X =  -36.989  mm,	Y =   -302.342  mm,	Z =   -251.166  mm,
	W =  90.000 deg,	P =   0.000 deg,	R =   90.000 deg
};
P[2641]{
   GP1:
	UF : 0, UT : 6,		CONFIG : 'N U T, 0, 0, 0',
	X =  -38.238  mm,	Y =   -303.009  mm,	Z =   -251.039  mm,
	W =  90.000 deg,	P =   0.000 deg,	R =   90.000 deg
};
P[2642]{
   GP1:
	UF : 0, UT : 6,		CONFIG : 'N U T, 0, 0, 0',
	X =  -39.472  mm,	Y =   -303.837  mm,	Z =   -251.317  mm,
	W =  90.000 deg,	P =   0.000 deg,	R =   90.000 deg
};
P[2643]{
   GP1:
	UF : 0, UT : 6,		CONFIG : 'N U T, 0, 0, 0',
	X =  -43.736  mm,	Y =   -306.357  mm,	Z =   -251.458  mm,
	W =  90.000 deg,	P =   0.000 deg,	R =   90.000 deg
};
P[2644]{
   GP1:
	UF : 0, UT : 6,		CONFIG : 'N U T, 0, 0, 0',
	X =  -44.598  mm,	Y =   -306.811  mm,	Z =   -251.353  mm,
	W =  90.000 deg,	P =   0.000 deg,	R =   90.000 deg
};
P[2645]{
   GP1:
	UF : 0, UT : 6,		CONFIG : 'N U T, 0, 0, 0',
	X =  -45.460  mm,	Y =   -307.251  mm,	Z =   -251.213  mm,
	W =  90.000 deg,	P =   0.000 deg,	R =   90.000 deg
};
P[2646]{
   GP1:
	UF : 0, UT : 6,		CONFIG : 'N U T, 0, 0, 0',
	X =  -46.368  mm,	Y =   -307.742  mm,	Z =   -251.131  mm,
	W =  90.000 deg,	P =   0.000 deg,	R =   90.000 deg
};
P[2647]{
   GP1:
	UF : 0, UT : 6,		CONFIG : 'N U T, 0, 0, 0',
	X =  -47.190  mm,	Y =   -308.373  mm,	Z =   -251.511  mm,
	W =  90.000 deg,	P =   0.000 deg,	R =   90.000 deg
};
P[2648]{
   GP1:
	UF : 0, UT : 6,		CONFIG : 'N U T, 0, 0, 0',
	X =  -47.954  mm,	Y =   -308.781  mm,	Z =   -251.429  mm,
	W =  90.000 deg,	P =   0.000 deg,	R =   90.000 deg
};
P[2649]{
   GP1:
	UF : 0, UT : 6,		CONFIG : 'N U T, 0, 0, 0',
	X =  -48.975  mm,	Y =   -309.322  mm,	Z =   -251.314  mm,
	W =  90.000 deg,	P =   0.000 deg,	R =   90.000 deg
};
P[2650]{
   GP1:
	UF : 0, UT : 6,		CONFIG : 'N U T, 0, 0, 0',
	X =  -52.883  mm,	Y =   -311.524  mm,	Z =   -251.180  mm,
	W =  90.000 deg,	P =   0.000 deg,	R =   90.000 deg
};
P[2651]{
   GP1:
	UF : 0, UT : 6,		CONFIG : 'N U T, 0, 0, 0',
	X =  -54.913  mm,	Y =   -312.783  mm,	Z =   -251.392  mm,
	W =  90.000 deg,	P =   0.000 deg,	R =   90.000 deg
};
P[2652]{
   GP1:
	UF : 0, UT : 6,		CONFIG : 'N U T, 0, 0, 0',
	X =  -59.258  mm,	Y =   -315.340  mm,	Z =   -251.507  mm,
	W =  90.000 deg,	P =   0.000 deg,	R =   90.000 deg
};
P[2653]{
   GP1:
	UF : 0, UT : 6,		CONFIG : 'N U T, 0, 0, 0',
	X =  -64.226  mm,	Y =   -318.100  mm,	Z =   -251.245  mm,
	W =  90.000 deg,	P =   0.000 deg,	R =   90.000 deg
};
P[2654]{
   GP1:
	UF : 0, UT : 6,		CONFIG : 'N U T, 0, 0, 0',
	X =  -65.377  mm,	Y =   -318.836  mm,	Z =   -251.420  mm,
	W =  90.000 deg,	P =   0.000 deg,	R =   90.000 deg
};
P[2655]{
   GP1:
	UF : 0, UT : 6,		CONFIG : 'N U T, 0, 0, 0',
	X =  -66.318  mm,	Y =   -319.335  mm,	Z =   -251.309  mm,
	W =  90.000 deg,	P =   0.000 deg,	R =   90.000 deg
};
P[2656]{
   GP1:
	UF : 0, UT : 6,		CONFIG : 'N U T, 0, 0, 0',
	X =  -68.403  mm,	Y =   -320.602  mm,	Z =   -251.463  mm,
	W =  90.000 deg,	P =   0.000 deg,	R =   90.000 deg
};
P[2657]{
   GP1:
	UF : 0, UT : 6,		CONFIG : 'N U T, 0, 0, 0',
	X =  -70.633  mm,	Y =   -321.902  mm,	Z =   -251.494  mm,
	W =  90.000 deg,	P =   0.000 deg,	R =   90.000 deg
};
P[2658]{
   GP1:
	UF : 0, UT : 6,		CONFIG : 'N U T, 0, 0, 0',
	X =  -73.090  mm,	Y =   -323.282  mm,	Z =   -251.400  mm,
	W =  90.000 deg,	P =   0.000 deg,	R =   90.000 deg
};
P[2659]{
   GP1:
	UF : 0, UT : 6,		CONFIG : 'N U T, 0, 0, 0',
	X =  -75.366  mm,	Y =   -324.482  mm,	Z =   -251.122  mm,
	W =  90.000 deg,	P =   0.000 deg,	R =   90.000 deg
};
P[2660]{
   GP1:
	UF : 0, UT : 6,		CONFIG : 'N U T, 0, 0, 0',
	X =  -77.217  mm,	Y =   -325.538  mm,	Z =   -251.093  mm,
	W =  90.000 deg,	P =   0.000 deg,	R =   90.000 deg
};
P[2661]{
   GP1:
	UF : 0, UT : 6,		CONFIG : 'N U T, 0, 0, 0',
	X =  -77.878  mm,	Y =   -326.030  mm,	Z =   -251.359  mm,
	W =  90.000 deg,	P =   0.000 deg,	R =   90.000 deg
};
P[2662]{
   GP1:
	UF : 0, UT : 6,		CONFIG : 'N U T, 0, 0, 0',
	X =  -81.229  mm,	Y =   -327.912  mm,	Z =   -251.231  mm,
	W =  90.000 deg,	P =   0.000 deg,	R =   90.000 deg
};
P[2663]{
   GP1:
	UF : 0, UT : 6,		CONFIG : 'N U T, 0, 0, 0',
	X =  -83.967  mm,	Y =   -329.568  mm,	Z =   -251.413  mm,
	W =  90.000 deg,	P =   0.000 deg,	R =   90.000 deg
};
P[2664]{
   GP1:
	UF : 0, UT : 6,		CONFIG : 'N U T, 0, 0, 0',
	X =  -86.936  mm,	Y =   -331.264  mm,	Z =   -251.371  mm,
	W =  90.000 deg,	P =   0.000 deg,	R =   90.000 deg
};
P[2665]{
   GP1:
	UF : 0, UT : 6,		CONFIG : 'N U T, 0, 0, 0',
	X =  -88.237  mm,	Y =   -332.062  mm,	Z =   -251.482  mm,
	W =  90.000 deg,	P =   0.000 deg,	R =   90.000 deg
};
